   1:  PR[GP1:91,2] = PR[GP1:90,2] + -0.839;
   1:L PR[91] 10mm/sec CNT100;
   1:  PR[GP1:91,1] = PR[GP1:90,1] + 35.563;
   1:  PR[GP1:91,2] = PR[GP1:90,2] + -0.395;
   1:L PR[91] 10mm/sec CNT100;
   1:  PR[GP1:91,1] = PR[GP1:90,1] + 35.190;
   1:  PR[GP1:91,2] = PR[GP1:90,2] + 2.914;
   1:L PR[91] 10mm/sec CNT100;
   1:  PR[GP1:91,1] = PR[GP1:90,1] + 34.179;
   1:  PR[GP1:91,2] = PR[GP1:90,2] + 6.099;
   1:L PR[91] 10mm/sec CNT100;
   1:  PR[GP1:91,1] = PR[GP1:90,1] + 32.535;
   1:  PR[GP1:91,2] = PR[GP1:90,2] + 9.023;
   1:L PR[91] 10mm/sec CNT100;
   1:  PR[GP1:91,1] = PR[GP1:90,1] + 30.321;
   1:  PR[GP1:91,2] = PR[GP1:90,2] + 11.577;
   1:L PR[91] 10mm/sec CNT100;
   1:  PR[GP1:91,1] = PR[GP1:90,1] + 27.624;
   1:  PR[GP1:91,2] = PR[GP1:90,2] + 13.659;
   1:L PR[91] 10mm/sec CNT100;
   1:  PR[GP1:91,1] = PR[GP1:90,1] + 25.039;
   1:  PR[GP1:91,2] = PR[GP1:90,2] + 14.946;
   1:L PR[91] 10mm/sec CNT100;
   1:  PR[GP1:91,1] = PR[GP1:90,1] + 24.543;
   1:  PR[GP1:91,2] = PR[GP1:90,2] + 15.184;
   1:L PR[91] 10mm/sec CNT100;
   1:  PR[GP1:91,1] = PR[GP1:90,1] + 21.112;
   1:  PR[GP1:91,2] = PR[GP1:90,2] + 16.090;
   1:L PR[91] 10mm/sec CNT100;
   1:  PR[GP1:91,1] = PR[GP1:90,1] + 17.539;
   1:  PR[GP1:91,2] = PR[GP1:90,2] + 16.343;
   1:L PR[91] 10mm/sec CNT100;
   1:  PR[GP1:91,1] = PR[GP1:90,1] + 16.151;
   1:  PR[GP1:91,2] = PR[GP1:90,2] + 16.185;
   1:L PR[91] 10mm/sec CNT100;
   1:  PR[GP1:91,1] = PR[GP1:90,1] + 13.927;
   1:  PR[GP1:91,2] = PR[GP1:90,2] + 15.922;
   1:L PR[91] 10mm/sec CNT100;
   1:  PR[GP1:91,1] = PR[GP1:90,1] + 10.426;
   1:  PR[GP1:91,2] = PR[GP1:90,2] + 14.850;
   1:L PR[91] 10mm/sec CNT100;
   1:  PR[GP1:91,1] = PR[GP1:90,1] + 7.184;
   1:  PR[GP1:91,2] = PR[GP1:90,2] + 13.161;
   1:L PR[91] 10mm/sec CNT100;
   1:  PR[GP1:91,1] = PR[GP1:90,1] + 4.339;
   1:  PR[GP1:91,2] = PR[GP1:90,2] + 10.940;
   1:L PR[91] 10mm/sec CNT100;
   1:  PR[GP1:91,1] = PR[GP1:90,1] + 2.001;
   1:  PR[GP1:91,2] = PR[GP1:90,2] + 8.245;
   1:L PR[91] 10mm/sec CNT100;
   1:  PR[GP1:91,1] = PR[GP1:90,1] + 1.503;
   1:  PR[GP1:91,2] = PR[GP1:90,2] + 7.522;
   1:L PR[91] 10mm/sec CNT100;
   1:  PR[GP1:91,1] = PR[GP1:90,1] + 1.266;
   1:  PR[GP1:91,2] = PR[GP1:90,2] + 7.119;
   1:L PR[91] 10mm/sec CNT100;
   1:  PR[GP1:91,1] = PR[GP1:90,1] + 0.739;
   1:  PR[GP1:91,2] = PR[GP1:90,2] + 6.549;
   1:L PR[91] 10mm/sec CNT100;
   1:  PR[GP1:91,1] = PR[GP1:90,1] + 0.420;
   1:  PR[GP1:91,2] = PR[GP1:90,2] + 6.165;
   1:L PR[91] 10mm/sec CNT100;
   1:  PR[GP1:91,1] = PR[GP1:90,1] + -0.128;
   1:  PR[GP1:91,2] = PR[GP1:90,2] + 5.978;
   1:L PR[91] 10mm/sec CNT100;
   1:  PR[GP1:91,1] = PR[GP1:90,1] + -0.975;
   1:  PR[GP1:91,2] = PR[GP1:90,2] + 5.799;
   1:L PR[91] 10mm/sec CNT100;
   1:  PR[GP1:91,1] = PR[GP1:90,1] + -2.276;
   1:  PR[GP1:91,2] = PR[GP1:90,2] + 6.339;
   1:L PR[91] 10mm/sec CNT100;
   1:  PR[GP1:91,1] = PR[GP1:90,1] + -3.093;
   1:  PR[GP1:91,2] = PR[GP1:90,2] + 7.226;
   1:L PR[91] 10mm/sec CNT100;
   1:  PR[GP1:91,1] = PR[GP1:90,1] + -3.176;
   1:  PR[GP1:91,2] = PR[GP1:90,2] + 7.385;
   1:L PR[91] 10mm/sec CNT100;
   1:  PR[GP1:91,1] = PR[GP1:90,1] + -4.802;
   1:  PR[GP1:91,2] = PR[GP1:90,2] + 9.594;
   1:L PR[91] 10mm/sec CNT100;
   1:  PR[GP1:91,1] = PR[GP1:90,1] + -5.353;
   1:  PR[GP1:91,2] = PR[GP1:90,2] + 10.305;
   1:L PR[91] 10mm/sec CNT100;
   1:  PR[GP1:91,1] = PR[GP1:90,1] + -6.810;
   1:  PR[GP1:91,2] = PR[GP1:90,2] + 11.631;
   1:L PR[91] 10mm/sec CNT100;
   1:  PR[GP1:91,1] = PR[GP1:90,1] + -8.065;
   1:  PR[GP1:91,2] = PR[GP1:90,2] + 12.724;
   1:L PR[91] 10mm/sec CNT100;
   1:  PR[GP1:91,1] = PR[GP1:90,1] + -9.145;
   1:  PR[GP1:91,2] = PR[GP1:90,2] + 13.374;
   1:L PR[91] 10mm/sec CNT100;
   1:  PR[GP1:91,1] = PR[GP1:90,1] + -11.190;
   1:  PR[GP1:91,2] = PR[GP1:90,2] + 14.553;
   1:L PR[91] 10mm/sec CNT100;
   1:  PR[GP1:91,1] = PR[GP1:90,1] + -14.602;
   1:  PR[GP1:91,2] = PR[GP1:90,2] + 15.736;
   1:L PR[91] 10mm/sec CNT100;
   1:  PR[GP1:91,1] = PR[GP1:90,1] + -17.903;
   1:  PR[GP1:91,2] = PR[GP1:90,2] + 16.202;
   1:L PR[91] 10mm/sec CNT100;
   1:  PR[GP1:91,1] = PR[GP1:90,1] + -18.257;
   1:  PR[GP1:91,2] = PR[GP1:90,2] + 16.208;
   1:L PR[91] 10mm/sec CNT100;
   1:  PR[GP1:91,1] = PR[GP1:90,1] + -21.180;
   1:  PR[GP1:91,2] = PR[GP1:90,2] + 16.036;
   1:L PR[91] 10mm/sec CNT100;
   1:  PR[GP1:91,1] = PR[GP1:90,1] + -21.987;
   1:  PR[GP1:91,2] = PR[GP1:90,2] + 15.880;
   1:L PR[91] 10mm/sec CNT100;
   1:  PR[GP1:91,1] = PR[GP1:90,1] + -24.427;
   1:  PR[GP1:91,2] = PR[GP1:90,2] + 15.235;
   1:L PR[91] 10mm/sec CNT100;
   1:  PR[GP1:91,1] = PR[GP1:90,1] + -25.526;
   1:  PR[GP1:91,2] = PR[GP1:90,2] + 14.770;
   1:L PR[91] 10mm/sec CNT100;
   1:  PR[GP1:91,1] = PR[GP1:90,1] + -27.498;
   1:  PR[GP1:91,2] = PR[GP1:90,2] + 13.796;
   1:L PR[91] 10mm/sec CNT100;
   1:  PR[GP1:91,1] = PR[GP1:90,1] + -28.704;
   1:  PR[GP1:91,2] = PR[GP1:90,2] + 12.949;
   1:L PR[91] 10mm/sec CNT100;
   1:  PR[GP1:91,1] = PR[GP1:90,1] + -30.246;
   1:  PR[GP1:91,2] = PR[GP1:90,2] + 11.752;
   1:L PR[91] 10mm/sec CNT100;
   1:  PR[GP1:91,1] = PR[GP1:90,1] + -31.379;
   1:  PR[GP1:91,2] = PR[GP1:90,2] + 10.524;
   1:L PR[91] 10mm/sec CNT100;
   1:  PR[GP1:91,1] = PR[GP1:90,1] + -32.532;
   1:  PR[GP1:91,2] = PR[GP1:90,2] + 9.173;
   1:L PR[91] 10mm/sec CNT100;
   1:  PR[GP1:91,1] = PR[GP1:90,1] + -33.440;
   1:  PR[GP1:91,2] = PR[GP1:90,2] + 7.630;
   1:L PR[91] 10mm/sec CNT100;
   1:  PR[GP1:91,1] = PR[GP1:90,1] + -34.248;
   1:  PR[GP1:91,2] = PR[GP1:90,2] + 6.164;
   1:L PR[91] 10mm/sec CNT100;
   1:  PR[GP1:91,1] = PR[GP1:90,1] + -34.824;
   1:  PR[GP1:91,2] = PR[GP1:90,2] + 4.418;
   1:L PR[91] 10mm/sec CNT100;
   1:  PR[GP1:91,1] = PR[GP1:90,1] + -35.313;
   1:  PR[GP1:91,2] = PR[GP1:90,2] + 2.861;
   1:L PR[91] 10mm/sec CNT100;
   1:  PR[GP1:91,1] = PR[GP1:90,1] + -35.500;
   1:  PR[GP1:91,2] = PR[GP1:90,2] + 1.034;
   1:L PR[91] 10mm/sec CNT100;
   1:  PR[GP1:91,1] = PR[GP1:90,1] + -35.737;
   1:  PR[GP1:91,2] = PR[GP1:90,2] + -0.426;
   1:L PR[91] 10mm/sec CNT100;
   1:  PR[GP1:91,1] = PR[GP1:90,1] + -35.748;
   1:  PR[GP1:91,2] = PR[GP1:90,2] + -0.547;
   1:L PR[91] 10mm/sec CNT100;
   1:  PR[GP1:91,1] = PR[GP1:90,1] + -35.460;
   1:  PR[GP1:91,2] = PR[GP1:90,2] + -2.299;
   1:L PR[91] 10mm/sec CNT100;
   1:  PR[GP1:91,1] = PR[GP1:90,1] + -35.263;
   1:  PR[GP1:91,2] = PR[GP1:90,2] + -4.065;
   1:L PR[91] 10mm/sec CNT100;
   1:  PR[GP1:91,1] = PR[GP1:90,1] + -34.667;
   1:  PR[GP1:91,2] = PR[GP1:90,2] + -5.939;
   1:L PR[91] 10mm/sec CNT100;
   1:  PR[GP1:91,1] = PR[GP1:90,1] + -34.192;
   1:  PR[GP1:91,2] = PR[GP1:90,2] + -7.356;
   1:L PR[91] 10mm/sec CNT100;
   1:  PR[GP1:91,1] = PR[GP1:90,1] + -33.095;
   1:  PR[GP1:91,2] = PR[GP1:90,2] + -9.301;
   1:L PR[91] 10mm/sec CNT100;
   1:  PR[GP1:91,1] = PR[GP1:90,1] + -32.472;
   1:  PR[GP1:91,2] = PR[GP1:90,2] + -10.348;
   1:L PR[91] 10mm/sec CNT100;
   1:  PR[GP1:91,1] = PR[GP1:90,1] + -30.781;
   1:  PR[GP1:91,2] = PR[GP1:90,2] + -12.296;
   1:L PR[91] 10mm/sec CNT100;
   1:  PR[GP1:91,1] = PR[GP1:90,1] + -30.208;
   1:  PR[GP1:91,2] = PR[GP1:90,2] + -12.915;
   1:L PR[91] 10mm/sec CNT100;
   1:  PR[GP1:91,1] = PR[GP1:90,1] + -27.823;
   1:  PR[GP1:91,2] = PR[GP1:90,2] + -14.750;
   1:L PR[91] 10mm/sec CNT100;
   1:  PR[GP1:91,1] = PR[GP1:90,1] + -27.525;
   1:  PR[GP1:91,2] = PR[GP1:90,2] + -14.960;
   1:L PR[91] 10mm/sec CNT100;
   1:  PR[GP1:91,1] = PR[GP1:90,1] + -24.458;
   1:  PR[GP1:91,2] = PR[GP1:90,2] + -16.461;
   1:L PR[91] 10mm/sec CNT100;
   1:  PR[GP1:91,1] = PR[GP1:90,1] + -24.049;
   1:  PR[GP1:91,2] = PR[GP1:90,2] + -16.598;
   1:  PR[GP1:91,3] = PR[GP1:90,3] + 16.500;
   1:L PR[91] 10mm/sec CNT100;
   1:  PR[GP1:91,1] = PR[GP1:90,1] + -21.809;
   1:  PR[GP1:91,2] = PR[GP1:90,2] + -17.202;
   1:L PR[91] 10mm/sec CNT100;
   1:  PR[GP1:91,1] = PR[GP1:90,1] + -20.477;
   1:  PR[GP1:91,2] = PR[GP1:90,2] + -17.522;
   1:L PR[91] 10mm/sec CNT100;
   1:  PR[GP1:91,1] = PR[GP1:90,1] + -18.846;
   1:  PR[GP1:91,2] = PR[GP1:90,2] + -17.637;
   1:L PR[91] 10mm/sec CNT100;
   1:  PR[GP1:91,1] = PR[GP1:90,1] + -16.756;
   1:  PR[GP1:91,2] = PR[GP1:90,2] + -17.718;
   1:L PR[91] 10mm/sec CNT100;
   1:  PR[GP1:91,1] = PR[GP1:90,1] + -15.910;
   1:  PR[GP1:91,2] = PR[GP1:90,2] + -17.613;
   1:L PR[91] 10mm/sec CNT100;
   1:  PR[GP1:91,1] = PR[GP1:90,1] + -13.050;
   1:  PR[GP1:91,2] = PR[GP1:90,2] + -17.151;
   1:L PR[91] 10mm/sec CNT100;
   1:  PR[GP1:91,1] = PR[GP1:90,1] + -10.065;
   1:  PR[GP1:91,2] = PR[GP1:90,2] + -16.120;
   1:L PR[91] 10mm/sec CNT100;
   1:  PR[GP1:91,1] = PR[GP1:90,1] + -9.281;
   1:  PR[GP1:91,2] = PR[GP1:90,2] + -15.790;
   1:L PR[91] 10mm/sec CNT100;
   1:  PR[GP1:91,1] = PR[GP1:90,1] + -7.395;
   1:  PR[GP1:91,2] = PR[GP1:90,2] + -14.673;
   1:L PR[91] 10mm/sec CNT100;
   1:  PR[GP1:91,1] = PR[GP1:90,1] + -5.918;
   1:  PR[GP1:91,2] = PR[GP1:90,2] + -13.640;
   1:L PR[91] 10mm/sec CNT100;
   1:  PR[GP1:91,1] = PR[GP1:90,1] + -5.000;
   1:  PR[GP1:91,2] = PR[GP1:90,2] + -12.787;
   1:L PR[91] 10mm/sec CNT100;
   1:  PR[GP1:91,1] = PR[GP1:90,1] + -3.184;
   1:  PR[GP1:91,2] = PR[GP1:90,2] + -10.770;
   1:L PR[91] 10mm/sec CNT100;
   1:  PR[GP1:91,1] = PR[GP1:90,1] + -2.909;
   1:  PR[GP1:91,2] = PR[GP1:90,2] + -10.366;
   1:L PR[91] 10mm/sec CNT100;
   1:  PR[GP1:91,1] = PR[GP1:90,1] + -2.225;
   1:  PR[GP1:91,2] = PR[GP1:90,2] + -9.700;
   1:L PR[91] 10mm/sec CNT100;
   1:  PR[GP1:91,1] = PR[GP1:90,1] + -1.965;
   1:  PR[GP1:91,2] = PR[GP1:90,2] + -9.545;
   1:L PR[91] 10mm/sec CNT100;
   1:  PR[GP1:91,1] = PR[GP1:90,1] + -1.033;
   1:  PR[GP1:91,2] = PR[GP1:90,2] + -9.287;
   1:L PR[91] 10mm/sec CNT100;
   1:  PR[GP1:91,1] = PR[GP1:90,1] + -0.752;
   1:  PR[GP1:91,2] = PR[GP1:90,2] + -9.306;
   1:L PR[91] 10mm/sec CNT100;
   1:  PR[GP1:91,1] = PR[GP1:90,1] + 0.181;
   1:  PR[GP1:91,2] = PR[GP1:90,2] + -9.570;
   1:L PR[91] 10mm/sec CNT100;
   1:  PR[GP1:91,1] = PR[GP1:90,1] + 0.446;
   1:  PR[GP1:91,2] = PR[GP1:90,2] + -9.766;
   1:L PR[91] 10mm/sec CNT100;
   1:  PR[GP1:91,1] = PR[GP1:90,1] + 1.063;
   1:  PR[GP1:91,2] = PR[GP1:90,2] + -10.427;
   1:L PR[91] 10mm/sec CNT100;
   1:  PR[GP1:91,1] = PR[GP1:90,1] + 1.209;
   1:  PR[GP1:91,2] = PR[GP1:90,2] + -10.623;
   1:L PR[91] 10mm/sec CNT100;
   1:  PR[GP1:91,1] = PR[GP1:90,1] + 2.802;
   1:  PR[GP1:91,2] = PR[GP1:90,2] + -12.531;
   1:L PR[91] 10mm/sec CNT100;
   1:  PR[GP1:91,1] = PR[GP1:90,1] + 3.060;
   1:  PR[GP1:91,2] = PR[GP1:90,2] + -12.778;
   1:L PR[91] 10mm/sec CNT100;
   1:  PR[GP1:91,1] = PR[GP1:90,1] + 4.730;
   1:  PR[GP1:91,2] = PR[GP1:90,2] + -14.227;
   1:L PR[91] 10mm/sec CNT100;
   1:  PR[GP1:91,1] = PR[GP1:90,1] + 5.384;
   1:  PR[GP1:91,2] = PR[GP1:90,2] + -14.675;
   1:L PR[91] 10mm/sec CNT100;
   1:  PR[GP1:91,1] = PR[GP1:90,1] + 6.911;
   1:  PR[GP1:91,2] = PR[GP1:90,2] + -15.628;
   1:L PR[91] 10mm/sec CNT100;
   1:  PR[GP1:91,1] = PR[GP1:90,1] + 8.184;
   1:  PR[GP1:91,2] = PR[GP1:90,2] + -16.230;
   1:L PR[91] 10mm/sec CNT100;
   1:  PR[GP1:91,1] = PR[GP1:90,1] + 9.302;
   1:  PR[GP1:91,2] = PR[GP1:90,2] + -16.710;
   1:L PR[91] 10mm/sec CNT100;
   1:  PR[GP1:91,1] = PR[GP1:90,1] + 11.435;
   1:  PR[GP1:91,2] = PR[GP1:90,2] + -17.342;
   1:L PR[91] 10mm/sec CNT100;
   1:  PR[GP1:91,1] = PR[GP1:90,1] + 11.858;
   1:  PR[GP1:91,2] = PR[GP1:90,2] + -17.453;
   1:L PR[91] 10mm/sec CNT100;
   1:  PR[GP1:91,1] = PR[GP1:90,1] + 13.231;
   1:  PR[GP1:91,2] = PR[GP1:90,2] + -17.645;
   1:L PR[91] 10mm/sec CNT100;
   1:  PR[GP1:91,1] = PR[GP1:90,1] + 14.565;
   1:  PR[GP1:91,2] = PR[GP1:90,2] + -17.853;
   1:L PR[91] 10mm/sec CNT100;
   1:  PR[GP1:91,1] = PR[GP1:90,1] + 17.338;
   1:  PR[GP1:91,2] = PR[GP1:90,2] + -17.894;
   1:L PR[91] 10mm/sec CNT100;
   1:  PR[GP1:91,1] = PR[GP1:90,1] + 20.128;
   1:  PR[GP1:91,2] = PR[GP1:90,2] + -17.557;
   1:L PR[91] 10mm/sec CNT100;
   1:  PR[GP1:91,1] = PR[GP1:90,1] + 22.900;
   1:  PR[GP1:91,2] = PR[GP1:90,2] + -16.831;
   1:L PR[91] 10mm/sec CNT100;
   1:  PR[GP1:91,1] = PR[GP1:90,1] + 25.555;
   1:  PR[GP1:91,2] = PR[GP1:90,2] + -15.714;
   1:L PR[91] 10mm/sec CNT100;
   1:  PR[GP1:91,1] = PR[GP1:90,1] + 27.990;
   1:  PR[GP1:91,2] = PR[GP1:90,2] + -14.238;
   1:L PR[91] 10mm/sec CNT100;
   1:  PR[GP1:91,1] = PR[GP1:90,1] + 30.137;
   1:  PR[GP1:91,2] = PR[GP1:90,2] + -12.447;
   1:L PR[91] 10mm/sec CNT100;
   1:  PR[GP1:91,1] = PR[GP1:90,1] + 31.915;
   1:  PR[GP1:91,2] = PR[GP1:90,2] + -10.393;
   1:L PR[91] 10mm/sec CNT100;
   1:  PR[GP1:91,1] = PR[GP1:90,1] + 33.342;
   1:  PR[GP1:91,2] = PR[GP1:90,2] + -8.106;
   1:L PR[91] 10mm/sec CNT100;
   1:  PR[GP1:91,1] = PR[GP1:90,1] + 34.386;
   1:  PR[GP1:91,2] = PR[GP1:90,2] + -5.644;
   1:L PR[91] 10mm/sec CNT100;
   1:  PR[GP1:91,1] = PR[GP1:90,1] + 35.021;
   1:  PR[GP1:91,2] = PR[GP1:90,2] + -3.065;
   1:L PR[91] 10mm/sec CNT100;
   1:  PR[GP1:91,1] = PR[GP1:90,1] + 35.141;
   1:  PR[GP1:91,2] = PR[GP1:90,2] + -1.599;
   1:L PR[91] 10mm/sec CNT100;
   1:  PR[GP1:91,1] = PR[GP1:90,1] + 35.273;
   1:  PR[GP1:91,2] = PR[GP1:90,2] + -0.425;
   1:L PR[91] 10mm/sec CNT100;
   1:  PR[GP1:91,1] = PR[GP1:90,1] + 34.888;
   1:  PR[GP1:91,2] = PR[GP1:90,2] + 2.885;
   1:L PR[91] 10mm/sec CNT100;
   1:  PR[GP1:91,1] = PR[GP1:90,1] + 33.871;
   1:  PR[GP1:91,2] = PR[GP1:90,2] + 6.072;
   1:L PR[91] 10mm/sec CNT100;
   1:  PR[GP1:91,1] = PR[GP1:90,1] + 32.223;
   1:  PR[GP1:91,2] = PR[GP1:90,2] + 8.997;
   1:L PR[91] 10mm/sec CNT100;
   1:  PR[GP1:91,1] = PR[GP1:90,1] + 30.005;
   1:  PR[GP1:91,2] = PR[GP1:90,2] + 11.551;
   1:L PR[91] 10mm/sec CNT100;
   1:  PR[GP1:91,1] = PR[GP1:90,1] + 28.164;
   1:  PR[GP1:91,2] = PR[GP1:90,2] + 12.971;
   1:L PR[91] 10mm/sec CNT100;
   1:  PR[GP1:91,1] = PR[GP1:90,1] + 27.290;
   1:  PR[GP1:91,2] = PR[GP1:90,2] + 13.625;
   1:L PR[91] 10mm/sec CNT100;
   1:  PR[GP1:91,1] = PR[GP1:90,1] + 24.125;
   1:  PR[GP1:91,2] = PR[GP1:90,2] + 15.144;
   1:L PR[91] 10mm/sec CNT100;
   1:  PR[GP1:91,1] = PR[GP1:90,1] + 20.701;
   1:  PR[GP1:91,2] = PR[GP1:90,2] + 16.048;
   1:L PR[91] 10mm/sec CNT100;
   1:  PR[GP1:91,1] = PR[GP1:90,1] + 17.093;
   1:  PR[GP1:91,2] = PR[GP1:90,2] + 16.290;
   1:L PR[91] 10mm/sec CNT100;
   1:  PR[GP1:91,1] = PR[GP1:90,1] + 13.444;
   1:  PR[GP1:91,2] = PR[GP1:90,2] + 15.859;
   1:L PR[91] 10mm/sec CNT100;
   1:  PR[GP1:91,1] = PR[GP1:90,1] + 9.932;
   1:  PR[GP1:91,2] = PR[GP1:90,2] + 14.773;
   1:L PR[91] 10mm/sec CNT100;
   1:  PR[GP1:91,1] = PR[GP1:90,1] + 6.681;
   1:  PR[GP1:91,2] = PR[GP1:90,2] + 13.083;
   1:L PR[91] 10mm/sec CNT100;
   1:  PR[GP1:91,1] = PR[GP1:90,1] + 3.849;
   1:  PR[GP1:91,2] = PR[GP1:90,2] + 10.848;
   1:L PR[91] 10mm/sec CNT100;
   1:  PR[GP1:91,1] = PR[GP1:90,1] + 1.504;
   1:  PR[GP1:91,2] = PR[GP1:90,2] + 8.159;
   1:L PR[91] 10mm/sec CNT100;
   1:  PR[GP1:91,1] = PR[GP1:90,1] + 1.159;
   1:  PR[GP1:91,2] = PR[GP1:90,2] + 7.659;
   1:L PR[91] 10mm/sec CNT100;
   1:  PR[GP1:91,1] = PR[GP1:90,1] + 0.530;
   1:  PR[GP1:91,2] = PR[GP1:90,2] + 7.106;
   1:L PR[91] 10mm/sec CNT100;
   1:  PR[GP1:91,1] = PR[GP1:90,1] + 0.267;
   1:  PR[GP1:91,2] = PR[GP1:90,2] + 6.814;
   1:L PR[91] 10mm/sec CNT100;
   1:  PR[GP1:91,1] = PR[GP1:90,1] + -1.097;
   1:  PR[GP1:91,2] = PR[GP1:90,2] + 6.515;
   1:L PR[91] 10mm/sec CNT100;
   1:  PR[GP1:91,1] = PR[GP1:90,1] + -1.473;
   1:  PR[GP1:91,2] = PR[GP1:90,2] + 6.676;
   1:L PR[91] 10mm/sec CNT100;
   1:  PR[GP1:91,1] = PR[GP1:90,1] + -2.323;
   1:  PR[GP1:91,2] = PR[GP1:90,2] + 6.945;
   1:L PR[91] 10mm/sec CNT100;
   1:  PR[GP1:91,1] = PR[GP1:90,1] + -3.014;
   1:  PR[GP1:91,2] = PR[GP1:90,2] + 7.674;
   1:L PR[91] 10mm/sec CNT100;
   1:  PR[GP1:91,1] = PR[GP1:90,1] + -4.937;
   1:  PR[GP1:91,2] = PR[GP1:90,2] + 10.131;
   1:L PR[91] 10mm/sec CNT100;
   1:  PR[GP1:91,1] = PR[GP1:90,1] + -7.022;
   1:  PR[GP1:91,2] = PR[GP1:90,2] + 12.028;
   1:L PR[91] 10mm/sec CNT100;
   1:  PR[GP1:91,1] = PR[GP1:90,1] + -7.655;
   1:  PR[GP1:91,2] = PR[GP1:90,2] + 12.579;
   1:L PR[91] 10mm/sec CNT100;
   1:  PR[GP1:91,1] = PR[GP1:90,1] + -9.399;
   1:  PR[GP1:91,2] = PR[GP1:90,2] + 13.630;
   1:L PR[91] 10mm/sec CNT100;
   1:  PR[GP1:91,1] = PR[GP1:90,1] + -10.792;
   1:  PR[GP1:91,2] = PR[GP1:90,2] + 14.432;
   1:L PR[91] 10mm/sec CNT100;
   1:  PR[GP1:91,1] = PR[GP1:90,1] + -12.052;
   1:  PR[GP1:91,2] = PR[GP1:90,2] + 14.889;
   1:L PR[91] 10mm/sec CNT100;
   1:  PR[GP1:91,1] = PR[GP1:90,1] + -14.210;
   1:  PR[GP1:91,2] = PR[GP1:90,2] + 15.629;
   1:L PR[91] 10mm/sec CNT100;
   1:  PR[GP1:91,1] = PR[GP1:90,1] + -17.771;
   1:  PR[GP1:91,2] = PR[GP1:90,2] + 16.139;
   1:L PR[91] 10mm/sec CNT100;
   1:  PR[GP1:91,1] = PR[GP1:90,1] + -21.225;
   1:  PR[GP1:91,2] = PR[GP1:90,2] + 15.950;
   1:L PR[91] 10mm/sec CNT100;
   1:  PR[GP1:91,1] = PR[GP1:90,1] + -21.354;
   1:  PR[GP1:91,2] = PR[GP1:90,2] + 15.925;
   1:L PR[91] 10mm/sec CNT100;
   1:  PR[GP1:91,1] = PR[GP1:90,1] + -24.418;
   1:  PR[GP1:91,2] = PR[GP1:90,2] + 15.116;
   1:L PR[91] 10mm/sec CNT100;
   1:  PR[GP1:91,1] = PR[GP1:90,1] + -24.918;
   1:  PR[GP1:91,2] = PR[GP1:90,2] + 14.903;
   1:L PR[91] 10mm/sec CNT100;
   1:  PR[GP1:91,1] = PR[GP1:90,1] + -27.439;
   1:  PR[GP1:91,2] = PR[GP1:90,2] + 13.659;
   1:L PR[91] 10mm/sec CNT100;
   1:  PR[GP1:91,1] = PR[GP1:90,1] + -28.140;
   1:  PR[GP1:91,2] = PR[GP1:90,2] + 13.167;
   1:L PR[91] 10mm/sec CNT100;
   1:  PR[GP1:91,1] = PR[GP1:90,1] + -30.142;
   1:  PR[GP1:91,2] = PR[GP1:90,2] + 11.612;
   1:L PR[91] 10mm/sec CNT100;
   1:  PR[GP1:91,1] = PR[GP1:90,1] + -30.873;
   1:  PR[GP1:91,2] = PR[GP1:90,2] + 10.820;
   1:L PR[91] 10mm/sec CNT100;
   1:  PR[GP1:91,1] = PR[GP1:90,1] + -32.392;
   1:  PR[GP1:91,2] = PR[GP1:90,2] + 9.041;
   1:L PR[91] 10mm/sec CNT100;
   1:  PR[GP1:91,1] = PR[GP1:90,1] + -33.008;
   1:  PR[GP1:91,2] = PR[GP1:90,2] + 7.994;
   1:L PR[91] 10mm/sec CNT100;
   1:  PR[GP1:91,1] = PR[GP1:90,1] + -34.079;
   1:  PR[GP1:91,2] = PR[GP1:90,2] + 6.050;
   1:L PR[91] 10mm/sec CNT100;
   1:  PR[GP1:91,1] = PR[GP1:90,1] + -34.479;
   1:  PR[GP1:91,2] = PR[GP1:90,2] + 4.838;
   1:L PR[91] 10mm/sec CNT100;
   1:  PR[GP1:91,1] = PR[GP1:90,1] + -35.129;
   1:  PR[GP1:91,2] = PR[GP1:90,2] + 2.771;
   1:L PR[91] 10mm/sec CNT100;
   1:  PR[GP1:91,1] = PR[GP1:90,1] + -35.259;
   1:  PR[GP1:91,2] = PR[GP1:90,2] + 1.496;
   1:L PR[91] 10mm/sec CNT100;
   1:  PR[GP1:91,1] = PR[GP1:90,1] + -35.426;
   1:  PR[GP1:91,2] = PR[GP1:90,2] + 0.467;
   1:L PR[91] 10mm/sec CNT100;
   1:  PR[GP1:91,1] = PR[GP1:90,1] + -35.526;
   1:  PR[GP1:91,2] = PR[GP1:90,2] + -0.621;
   1:L PR[91] 10mm/sec CNT100;
   1:  PR[GP1:91,1] = PR[GP1:90,1] + -35.330;
   1:  PR[GP1:91,2] = PR[GP1:90,2] + -1.808;
   1:L PR[91] 10mm/sec CNT100;
   1:  PR[GP1:91,1] = PR[GP1:90,1] + -35.074;
   1:  PR[GP1:91,2] = PR[GP1:90,2] + -4.102;
   1:L PR[91] 10mm/sec CNT100;
   1:  PR[GP1:91,1] = PR[GP1:90,1] + -34.300;
   1:  PR[GP1:91,2] = PR[GP1:90,2] + -6.541;
   1:L PR[91] 10mm/sec CNT100;
   1:  PR[GP1:91,1] = PR[GP1:90,1] + -34.023;
   1:  PR[GP1:91,2] = PR[GP1:90,2] + -7.366;
   1:L PR[91] 10mm/sec CNT100;
   1:  PR[GP1:91,1] = PR[GP1:90,1] + -32.618;
   1:  PR[GP1:91,2] = PR[GP1:90,2] + -9.858;
   1:L PR[91] 10mm/sec CNT100;
   1:  PR[GP1:91,1] = PR[GP1:90,1] + -32.333;
   1:  PR[GP1:91,2] = PR[GP1:90,2] + -10.338;
   1:L PR[91] 10mm/sec CNT100;
   1:  PR[GP1:91,1] = PR[GP1:90,1] + -30.204;
   1:  PR[GP1:91,2] = PR[GP1:90,2] + -12.789;
   1:L PR[91] 10mm/sec CNT100;
   1:  PR[GP1:91,1] = PR[GP1:90,1] + -30.110;
   1:  PR[GP1:91,2] = PR[GP1:90,2] + -12.891;
   1:L PR[91] 10mm/sec CNT100;
   1:  PR[GP1:91,1] = PR[GP1:90,1] + -27.320;
   1:  PR[GP1:91,2] = PR[GP1:90,2] + -15.014;
   1:L PR[91] 10mm/sec CNT100;
   1:  PR[GP1:91,1] = PR[GP1:90,1] + -24.722;
   1:  PR[GP1:91,2] = PR[GP1:90,2] + -16.288;
   1:L PR[91] 10mm/sec CNT100;
   1:  PR[GP1:91,1] = PR[GP1:90,1] + -23.632;
   1:  PR[GP1:91,2] = PR[GP1:90,2] + -16.737;
   1:  PR[GP1:91,3] = PR[GP1:90,3] + 17.600;
   1:L PR[91] 10mm/sec CNT100;
   1:  PR[GP1:91,1] = PR[GP1:90,1] + -22.073;
   1:  PR[GP1:91,2] = PR[GP1:90,2] + -17.157;
   1:L PR[91] 10mm/sec CNT100;
   1:  PR[GP1:91,1] = PR[GP1:90,1] + -20.031;
   1:  PR[GP1:91,2] = PR[GP1:90,2] + -17.648;
   1:L PR[91] 10mm/sec CNT100;
   1:  PR[GP1:91,1] = PR[GP1:90,1] + -19.162;
   1:  PR[GP1:91,2] = PR[GP1:90,2] + -17.710;
   1:L PR[91] 10mm/sec CNT100;
   1:  PR[GP1:91,1] = PR[GP1:90,1] + -16.282;
   1:  PR[GP1:91,2] = PR[GP1:90,2] + -17.821;
   1:L PR[91] 10mm/sec CNT100;
   1:  PR[GP1:91,1] = PR[GP1:90,1] + -13.121;
   1:  PR[GP1:91,2] = PR[GP1:90,2] + -17.389;
   1:L PR[91] 10mm/sec CNT100;
   1:  PR[GP1:91,1] = PR[GP1:90,1] + -12.278;
   1:  PR[GP1:91,2] = PR[GP1:90,2] + -17.222;
   1:L PR[91] 10mm/sec CNT100;
   1:  PR[GP1:91,1] = PR[GP1:90,1] + -10.225;
   1:  PR[GP1:91,2] = PR[GP1:90,2] + -16.518;
   1:L PR[91] 10mm/sec CNT100;
   1:  PR[GP1:91,1] = PR[GP1:90,1] + -8.447;
   1:  PR[GP1:91,2] = PR[GP1:90,2] + -15.769;
   1:L PR[91] 10mm/sec CNT100;
   1:  PR[GP1:91,1] = PR[GP1:90,1] + -7.521;
   1:  PR[GP1:91,2] = PR[GP1:90,2] + -15.220;
   1:L PR[91] 10mm/sec CNT100;
   1:  PR[GP1:91,1] = PR[GP1:90,1] + -5.098;
   1:  PR[GP1:91,2] = PR[GP1:90,2] + -13.526;
   1:L PR[91] 10mm/sec CNT100;
   1:  PR[GP1:91,1] = PR[GP1:90,1] + -4.779;
   1:  PR[GP1:91,2] = PR[GP1:90,2] + -13.184;
   1:L PR[91] 10mm/sec CNT100;
   1:  PR[GP1:91,1] = PR[GP1:90,1] + -2.747;
   1:  PR[GP1:91,2] = PR[GP1:90,2] + -11.110;
   1:L PR[91] 10mm/sec CNT100;
   1:  PR[GP1:91,1] = PR[GP1:90,1] + -2.284;
   1:  PR[GP1:91,2] = PR[GP1:90,2] + -10.666;
   1:L PR[91] 10mm/sec CNT100;
   1:  PR[GP1:91,1] = PR[GP1:90,1] + -1.776;
   1:  PR[GP1:91,2] = PR[GP1:90,2] + -10.363;
   1:L PR[91] 10mm/sec CNT100;
   1:  PR[GP1:91,1] = PR[GP1:90,1] + -1.082;
   1:  PR[GP1:91,2] = PR[GP1:90,2] + -10.171;
   1:L PR[91] 10mm/sec CNT100;
   1:  PR[GP1:91,1] = PR[GP1:90,1] + -0.525;
   1:  PR[GP1:91,2] = PR[GP1:90,2] + -10.209;
   1:L PR[91] 10mm/sec CNT100;
   1:  PR[GP1:91,1] = PR[GP1:90,1] + 0.158;
   1:  PR[GP1:91,2] = PR[GP1:90,2] + -10.402;
   1:L PR[91] 10mm/sec CNT100;
   1:  PR[GP1:91,1] = PR[GP1:90,1] + 0.712;
   1:  PR[GP1:91,2] = PR[GP1:90,2] + -10.812;
   1:L PR[91] 10mm/sec CNT100;
   1:  PR[GP1:91,1] = PR[GP1:90,1] + 0.851;
   1:  PR[GP1:91,2] = PR[GP1:90,2] + -11.005;
   1:L PR[91] 10mm/sec CNT100;
   1:  PR[GP1:91,1] = PR[GP1:90,1] + 1.058;
   1:  PR[GP1:91,2] = PR[GP1:90,2] + -11.227;
   1:L PR[91] 10mm/sec CNT100;
   1:  PR[GP1:91,1] = PR[GP1:90,1] + 2.039;
   1:  PR[GP1:91,2] = PR[GP1:90,2] + -12.391;
   1:L PR[91] 10mm/sec CNT100;
   1:  PR[GP1:91,1] = PR[GP1:90,1] + 2.398;
   1:  PR[GP1:91,2] = PR[GP1:90,2] + -12.782;
   1:L PR[91] 10mm/sec CNT100;
   1:  PR[GP1:91,1] = PR[GP1:90,1] + 4.390;
   1:  PR[GP1:91,2] = PR[GP1:90,2] + -14.508;
   1:L PR[91] 10mm/sec CNT100;
   1:  PR[GP1:91,1] = PR[GP1:90,1] + 6.605;
   1:  PR[GP1:91,2] = PR[GP1:90,2] + -15.893;
   1:L PR[91] 10mm/sec CNT100;
   1:  PR[GP1:91,1] = PR[GP1:90,1] + 7.051;
   1:  PR[GP1:91,2] = PR[GP1:90,2] + -16.104;
   1:L PR[91] 10mm/sec CNT100;
   1:  PR[GP1:91,1] = PR[GP1:90,1] + 9.006;
   1:  PR[GP1:91,2] = PR[GP1:90,2] + -16.943;
   1:L PR[91] 10mm/sec CNT100;
   1:  PR[GP1:91,1] = PR[GP1:90,1] + 10.197;
   1:  PR[GP1:91,2] = PR[GP1:90,2] + -17.296;
   1:L PR[91] 10mm/sec CNT100;
   1:  PR[GP1:91,1] = PR[GP1:90,1] + 11.566;
   1:  PR[GP1:91,2] = PR[GP1:90,2] + -17.656;
   1:L PR[91] 10mm/sec CNT100;
   1:  PR[GP1:91,1] = PR[GP1:90,1] + 13.741;
   1:  PR[GP1:91,2] = PR[GP1:90,2] + -17.960;
   1:L PR[91] 10mm/sec CNT100;
   1:  PR[GP1:91,1] = PR[GP1:90,1] + 14.236;
   1:  PR[GP1:91,2] = PR[GP1:90,2] + -18.015;
   1:L PR[91] 10mm/sec CNT100;
   1:  PR[GP1:91,1] = PR[GP1:90,1] + 15.625;
   1:  PR[GP1:91,2] = PR[GP1:90,2] + -18.006;
   1:L PR[91] 10mm/sec CNT100;
   1:  PR[GP1:91,1] = PR[GP1:90,1] + 17.004;
   1:  PR[GP1:91,2] = PR[GP1:90,2] + -18.020;
   1:L PR[91] 10mm/sec CNT100;
   1:  PR[GP1:91,1] = PR[GP1:90,1] + 19.780;
   1:  PR[GP1:91,2] = PR[GP1:90,2] + -17.663;
   1:L PR[91] 10mm/sec CNT100;
   1:  PR[GP1:91,1] = PR[GP1:90,1] + 22.509;
   1:  PR[GP1:91,2] = PR[GP1:90,2] + -16.928;
   1:L PR[91] 10mm/sec CNT100;
   1:  PR[GP1:91,1] = PR[GP1:90,1] + 25.143;
   1:  PR[GP1:91,2] = PR[GP1:90,2] + -15.812;
   1:L PR[91] 10mm/sec CNT100;
   1:  PR[GP1:91,1] = PR[GP1:90,1] + 27.585;
   1:  PR[GP1:91,2] = PR[GP1:90,2] + -14.329;
   1:L PR[91] 10mm/sec CNT100;
   1:  PR[GP1:91,1] = PR[GP1:90,1] + 29.750;
   1:  PR[GP1:91,2] = PR[GP1:90,2] + -12.524;
   1:L PR[91] 10mm/sec CNT100;
   1:  PR[GP1:91,1] = PR[GP1:90,1] + 31.588;
   1:  PR[GP1:91,2] = PR[GP1:90,2] + -10.446;
   1:L PR[91] 10mm/sec CNT100;
   1:  PR[GP1:91,1] = PR[GP1:90,1] + 33.034;
   1:  PR[GP1:91,2] = PR[GP1:90,2] + -8.151;
   1:L PR[91] 10mm/sec CNT100;
   1:  PR[GP1:91,1] = PR[GP1:90,1] + 34.075;
   1:  PR[GP1:91,2] = PR[GP1:90,2] + -5.686;
   1:L PR[91] 10mm/sec CNT100;
   1:  PR[GP1:91,1] = PR[GP1:90,1] + 34.708;
   1:  PR[GP1:91,2] = PR[GP1:90,2] + -3.102;
   1:L PR[91] 10mm/sec CNT100;
   1:  PR[GP1:91,1] = PR[GP1:90,1] + 34.769;
   1:  PR[GP1:91,2] = PR[GP1:90,2] + -2.359;
   1:L PR[91] 10mm/sec CNT100;
   1:  PR[GP1:91,1] = PR[GP1:90,1] + 34.868;
   1:  PR[GP1:91,2] = PR[GP1:90,2] + -1.475;
   1:L PR[91] 10mm/sec CNT100;
   1:  PR[GP1:91,1] = PR[GP1:90,1] + 34.947;
   1:  PR[GP1:91,2] = PR[GP1:90,2] + -0.465;
   1:L PR[91] 10mm/sec CNT100;
   1:  PR[GP1:91,1] = PR[GP1:90,1] + 34.749;
   1:  PR[GP1:91,2] = PR[GP1:90,2] + 1.466;
   1:L PR[91] 10mm/sec CNT100;
   1:  PR[GP1:91,1] = PR[GP1:90,1] + 34.585;
   1:  PR[GP1:91,2] = PR[GP1:90,2] + 2.856;
   1:L PR[91] 10mm/sec CNT100;
   1:  PR[GP1:91,1] = PR[GP1:90,1] + 33.563;
   1:  PR[GP1:91,2] = PR[GP1:90,2] + 6.045;
   1:L PR[91] 10mm/sec CNT100;
   1:  PR[GP1:91,1] = PR[GP1:90,1] + 31.912;
   1:  PR[GP1:91,2] = PR[GP1:90,2] + 8.968;
   1:L PR[91] 10mm/sec CNT100;
   1:  PR[GP1:91,1] = PR[GP1:90,1] + 29.647;
   1:  PR[GP1:91,2] = PR[GP1:90,2] + 11.512;
   1:L PR[91] 10mm/sec CNT100;
   1:  PR[GP1:91,1] = PR[GP1:90,1] + 26.874;
   1:  PR[GP1:91,2] = PR[GP1:90,2] + 13.585;
   1:L PR[91] 10mm/sec CNT100;
   1:  PR[GP1:91,1] = PR[GP1:90,1] + 23.708;
   1:  PR[GP1:91,2] = PR[GP1:90,2] + 15.103;
   1:L PR[91] 10mm/sec CNT100;
   1:  PR[GP1:91,1] = PR[GP1:90,1] + 21.814;
   1:  PR[GP1:91,2] = PR[GP1:90,2] + 15.603;
   1:L PR[91] 10mm/sec CNT100;
   1:  PR[GP1:91,1] = PR[GP1:90,1] + 20.251;
   1:  PR[GP1:91,2] = PR[GP1:90,2] + 15.995;
   1:L PR[91] 10mm/sec CNT100;
   1:  PR[GP1:91,1] = PR[GP1:90,1] + 16.603;
   1:  PR[GP1:91,2] = PR[GP1:90,2] + 16.224;
   1:L PR[91] 10mm/sec CNT100;
   1:  PR[GP1:91,1] = PR[GP1:90,1] + 13.589;
   1:  PR[GP1:91,2] = PR[GP1:90,2] + 15.869;
   1:L PR[91] 10mm/sec CNT100;
   1:  PR[GP1:91,1] = PR[GP1:90,1] + 12.958;
   1:  PR[GP1:91,2] = PR[GP1:90,2] + 15.788;
   1:L PR[91] 10mm/sec CNT100;
   1:  PR[GP1:91,1] = PR[GP1:90,1] + 9.434;
   1:  PR[GP1:91,2] = PR[GP1:90,2] + 14.689;
   1:L PR[91] 10mm/sec CNT100;
   1:  PR[GP1:91,1] = PR[GP1:90,1] + 6.191;
   1:  PR[GP1:91,2] = PR[GP1:90,2] + 12.993;
   1:L PR[91] 10mm/sec CNT100;
   1:  PR[GP1:91,1] = PR[GP1:90,1] + 3.357;
   1:  PR[GP1:91,2] = PR[GP1:90,2] + 10.754;
   1:L PR[91] 10mm/sec CNT100;
   1:  PR[GP1:91,1] = PR[GP1:90,1] + 1.082;
   1:  PR[GP1:91,2] = PR[GP1:90,2] + 8.169;
   1:L PR[91] 10mm/sec CNT100;
   1:  PR[GP1:91,1] = PR[GP1:90,1] + 0.172;
   1:  PR[GP1:91,2] = PR[GP1:90,2] + 7.329;
   1:L PR[91] 10mm/sec CNT100;
   1:  PR[GP1:91,1] = PR[GP1:90,1] + -0.803;
   1:  PR[GP1:91,2] = PR[GP1:90,2] + 7.136;
   1:L PR[91] 10mm/sec CNT100;
   1:  PR[GP1:91,1] = PR[GP1:90,1] + -1.222;
   1:  PR[GP1:91,2] = PR[GP1:90,2] + 7.098;
   1:L PR[91] 10mm/sec CNT100;
   1:  PR[GP1:91,1] = PR[GP1:90,1] + -1.703;
   1:  PR[GP1:91,2] = PR[GP1:90,2] + 7.333;
   1:L PR[91] 10mm/sec CNT100;
   1:  PR[GP1:91,1] = PR[GP1:90,1] + -2.383;
   1:  PR[GP1:91,2] = PR[GP1:90,2] + 7.548;
   1:L PR[91] 10mm/sec CNT100;
   1:  PR[GP1:91,1] = PR[GP1:90,1] + -2.969;
   1:  PR[GP1:91,2] = PR[GP1:90,2] + 8.153;
   1:L PR[91] 10mm/sec CNT100;
   1:  PR[GP1:91,1] = PR[GP1:90,1] + -4.270;
   1:  PR[GP1:91,2] = PR[GP1:90,2] + 9.798;
   1:L PR[91] 10mm/sec CNT100;
   1:  PR[GP1:91,1] = PR[GP1:90,1] + -4.896;
   1:  PR[GP1:91,2] = PR[GP1:90,2] + 10.399;
   1:L PR[91] 10mm/sec CNT100;
   1:  PR[GP1:91,1] = PR[GP1:90,1] + -7.244;
   1:  PR[GP1:91,2] = PR[GP1:90,2] + 12.433;
   1:L PR[91] 10mm/sec CNT100;
   1:  PR[GP1:91,1] = PR[GP1:90,1] + -9.654;
   1:  PR[GP1:91,2] = PR[GP1:90,2] + 13.885;
   1:L PR[91] 10mm/sec CNT100;
   1:  PR[GP1:91,1] = PR[GP1:90,1] + -10.389;
   1:  PR[GP1:91,2] = PR[GP1:90,2] + 14.309;
   1:L PR[91] 10mm/sec CNT100;
   1:  PR[GP1:91,1] = PR[GP1:90,1] + -12.324;
   1:  PR[GP1:91,2] = PR[GP1:90,2] + 15.010;
   1:L PR[91] 10mm/sec CNT100;
   1:  PR[GP1:91,1] = PR[GP1:90,1] + -13.823;
   1:  PR[GP1:91,2] = PR[GP1:90,2] + 15.524;
   1:L PR[91] 10mm/sec CNT100;
   1:  PR[GP1:91,1] = PR[GP1:90,1] + -15.203;
   1:  PR[GP1:91,2] = PR[GP1:90,2] + 15.738;
   1:L PR[91] 10mm/sec CNT100;
   1:  PR[GP1:91,1] = PR[GP1:90,1] + -17.392;
   1:  PR[GP1:91,2] = PR[GP1:90,2] + 16.044;
   1:L PR[91] 10mm/sec CNT100;
   1:  PR[GP1:91,1] = PR[GP1:90,1] + -20.959;
   1:  PR[GP1:91,2] = PR[GP1:90,2] + 15.864;
   1:L PR[91] 10mm/sec CNT100;
   1:  PR[GP1:91,1] = PR[GP1:90,1] + -24.373;
   1:  PR[GP1:91,2] = PR[GP1:90,2] + 15.002;
   1:L PR[91] 10mm/sec CNT100;
   1:  PR[GP1:91,1] = PR[GP1:90,1] + -27.380;
   1:  PR[GP1:91,2] = PR[GP1:90,2] + 13.522;
   1:L PR[91] 10mm/sec CNT100;
   1:  PR[GP1:91,1] = PR[GP1:90,1] + -27.575;
   1:  PR[GP1:91,2] = PR[GP1:90,2] + 13.385;
   1:L PR[91] 10mm/sec CNT100;
   1:  PR[GP1:91,1] = PR[GP1:90,1] + -30.039;
   1:  PR[GP1:91,2] = PR[GP1:90,2] + 11.472;
   1:L PR[91] 10mm/sec CNT100;
   1:  PR[GP1:91,1] = PR[GP1:90,1] + -30.368;
   1:  PR[GP1:91,2] = PR[GP1:90,2] + 11.116;
   1:L PR[91] 10mm/sec CNT100;
   1:  PR[GP1:91,1] = PR[GP1:90,1] + -32.251;
   1:  PR[GP1:91,2] = PR[GP1:90,2] + 8.910;
   1:L PR[91] 10mm/sec CNT100;
   1:  PR[GP1:91,1] = PR[GP1:90,1] + -32.576;
   1:  PR[GP1:91,2] = PR[GP1:90,2] + 8.357;
   1:L PR[91] 10mm/sec CNT100;
   1:  PR[GP1:91,1] = PR[GP1:90,1] + -33.909;
   1:  PR[GP1:91,2] = PR[GP1:90,2] + 5.939;
   1:L PR[91] 10mm/sec CNT100;
   1:  PR[GP1:91,1] = PR[GP1:90,1] + -34.944;
   1:  PR[GP1:91,2] = PR[GP1:90,2] + 2.680;
   1:L PR[91] 10mm/sec CNT100;
   1:  PR[GP1:91,1] = PR[GP1:90,1] + -35.018;
   1:  PR[GP1:91,2] = PR[GP1:90,2] + 1.958;
   1:L PR[91] 10mm/sec CNT100;
   1:  PR[GP1:91,1] = PR[GP1:90,1] + -35.115;
   1:  PR[GP1:91,2] = PR[GP1:90,2] + 1.360;
   1:L PR[91] 10mm/sec CNT100;
   1:  PR[GP1:91,1] = PR[GP1:90,1] + -35.303;
   1:  PR[GP1:91,2] = PR[GP1:90,2] + -0.695;
   1:L PR[91] 10mm/sec CNT100;
   1:  PR[GP1:91,1] = PR[GP1:90,1] + -35.201;
   1:  PR[GP1:91,2] = PR[GP1:90,2] + -1.317;
   1:L PR[91] 10mm/sec CNT100;
   1:  PR[GP1:91,1] = PR[GP1:90,1] + -34.886;
   1:  PR[GP1:91,2] = PR[GP1:90,2] + -4.138;
   1:L PR[91] 10mm/sec CNT100;
   1:  PR[GP1:91,1] = PR[GP1:90,1] + -33.851;
   1:  PR[GP1:91,2] = PR[GP1:90,2] + -7.381;
   1:L PR[91] 10mm/sec CNT100;
   1:  PR[GP1:91,1] = PR[GP1:90,1] + -32.319;
   1:  PR[GP1:91,2] = PR[GP1:90,2] + -10.099;
   1:L PR[91] 10mm/sec CNT100;
   1:  PR[GP1:91,1] = PR[GP1:90,1] + -32.182;
   1:  PR[GP1:91,2] = PR[GP1:90,2] + -10.334;
   1:L PR[91] 10mm/sec CNT100;
   1:  PR[GP1:91,1] = PR[GP1:90,1] + -29.816;
   1:  PR[GP1:91,2] = PR[GP1:90,2] + -12.989;
   1:L PR[91] 10mm/sec CNT100;
   1:  PR[GP1:91,1] = PR[GP1:90,1] + -27.613;
   1:  PR[GP1:91,2] = PR[GP1:90,2] + -14.661;
   1:L PR[91] 10mm/sec CNT100;
   1:  PR[GP1:91,1] = PR[GP1:90,1] + -26.936;
   1:  PR[GP1:91,2] = PR[GP1:90,2] + -15.155;
   1:L PR[91] 10mm/sec CNT100;
   1:  PR[GP1:91,1] = PR[GP1:90,1] + -24.919;
   1:  PR[GP1:91,2] = PR[GP1:90,2] + -16.144;
   1:L PR[91] 10mm/sec CNT100;
   1:  PR[GP1:91,1] = PR[GP1:90,1] + -23.216;
   1:  PR[GP1:91,2] = PR[GP1:90,2] + -16.876;
   1:  PR[GP1:91,3] = PR[GP1:90,3] + 18.700;
   1:L PR[91] 10mm/sec CNT100;
   1:  PR[GP1:91,1] = PR[GP1:90,1] + -22.336;
   1:  PR[GP1:91,2] = PR[GP1:90,2] + -17.113;
   1:L PR[91] 10mm/sec CNT100;
   1:  PR[GP1:91,1] = PR[GP1:90,1] + -19.589;
   1:  PR[GP1:91,2] = PR[GP1:90,2] + -17.774;
   1:L PR[91] 10mm/sec CNT100;
   1:  PR[GP1:91,1] = PR[GP1:90,1] + -16.314;
   1:  PR[GP1:91,2] = PR[GP1:90,2] + -17.952;
   1:L PR[91] 10mm/sec CNT100;
   1:  PR[GP1:91,1] = PR[GP1:90,1] + -15.570;
   1:  PR[GP1:91,2] = PR[GP1:90,2] + -17.955;
   1:L PR[91] 10mm/sec CNT100;
   1:  PR[GP1:91,1] = PR[GP1:90,1] + -13.285;
   1:  PR[GP1:91,2] = PR[GP1:90,2] + -17.647;
   1:L PR[91] 10mm/sec CNT100;
   1:  PR[GP1:91,1] = PR[GP1:90,1] + -11.478;
   1:  PR[GP1:91,2] = PR[GP1:90,2] + -17.290;
   1:L PR[91] 10mm/sec CNT100;
   1:  PR[GP1:91,1] = PR[GP1:90,1] + -10.385;
   1:  PR[GP1:91,2] = PR[GP1:90,2] + -16.915;
   1:L PR[91] 10mm/sec CNT100;
   1:  PR[GP1:91,1] = PR[GP1:90,1] + -7.623;
   1:  PR[GP1:91,2] = PR[GP1:90,2] + -15.751;
   1:L PR[91] 10mm/sec CNT100;
   1:  PR[GP1:91,1] = PR[GP1:90,1] + -4.850;
   1:  PR[GP1:91,2] = PR[GP1:90,2] + -13.992;
   1:L PR[91] 10mm/sec CNT100;
   1:  PR[GP1:91,1] = PR[GP1:90,1] + -3.957;
   1:  PR[GP1:91,2] = PR[GP1:90,2] + -13.266;
   1:L PR[91] 10mm/sec CNT100;
   1:  PR[GP1:91,1] = PR[GP1:90,1] + -2.604;
   1:  PR[GP1:91,2] = PR[GP1:90,2] + -11.876;
   1:L PR[91] 10mm/sec CNT100;
   1:  PR[GP1:91,1] = PR[GP1:90,1] + -2.342;
   1:  PR[GP1:91,2] = PR[GP1:90,2] + -11.631;
   1:L PR[91] 10mm/sec CNT100;
   1:  PR[GP1:91,1] = PR[GP1:90,1] + -1.587;
   1:  PR[GP1:91,2] = PR[GP1:90,2] + -11.181;
   1:L PR[91] 10mm/sec CNT100;
   1:  PR[GP1:91,1] = PR[GP1:90,1] + -1.131;
   1:  PR[GP1:91,2] = PR[GP1:90,2] + -11.055;
   1:L PR[91] 10mm/sec CNT100;
   1:  PR[GP1:91,1] = PR[GP1:90,1] + -0.299;
   1:  PR[GP1:91,2] = PR[GP1:90,2] + -11.112;
   1:L PR[91] 10mm/sec CNT100;
   1:  PR[GP1:91,1] = PR[GP1:90,1] + 0.136;
   1:  PR[GP1:91,2] = PR[GP1:90,2] + -11.235;
   1:L PR[91] 10mm/sec CNT100;
   1:  PR[GP1:91,1] = PR[GP1:90,1] + 0.944;
   1:  PR[GP1:91,2] = PR[GP1:90,2] + -11.833;
   1:L PR[91] 10mm/sec CNT100;
   1:  PR[GP1:91,1] = PR[GP1:90,1] + 1.103;
   1:  PR[GP1:91,2] = PR[GP1:90,2] + -12.055;
   1:L PR[91] 10mm/sec CNT100;
   1:  PR[GP1:91,1] = PR[GP1:90,1] + 1.583;
   1:  PR[GP1:91,2] = PR[GP1:90,2] + -12.592;
   1:L PR[91] 10mm/sec CNT100;
   1:  PR[GP1:91,1] = PR[GP1:90,1] + 1.969;
   1:  PR[GP1:91,2] = PR[GP1:90,2] + -12.993;
   1:L PR[91] 10mm/sec CNT100;
   1:  PR[GP1:91,1] = PR[GP1:90,1] + 3.562;
   1:  PR[GP1:91,2] = PR[GP1:90,2] + -14.381;
   1:L PR[91] 10mm/sec CNT100;
   1:  PR[GP1:91,1] = PR[GP1:90,1] + 4.090;
   1:  PR[GP1:91,2] = PR[GP1:90,2] + -14.802;
   1:L PR[91] 10mm/sec CNT100;
   1:  PR[GP1:91,1] = PR[GP1:90,1] + 6.295;
   1:  PR[GP1:91,2] = PR[GP1:90,2] + -16.153;
   1:L PR[91] 10mm/sec CNT100;
   1:  PR[GP1:91,1] = PR[GP1:90,1] + 8.700;
   1:  PR[GP1:91,2] = PR[GP1:90,2] + -17.173;
   1:L PR[91] 10mm/sec CNT100;
   1:  PR[GP1:91,1] = PR[GP1:90,1] + 11.275;
   1:  PR[GP1:91,2] = PR[GP1:90,2] + -17.859;
   1:L PR[91] 10mm/sec CNT100;
   1:  PR[GP1:91,1] = PR[GP1:90,1] + 12.406;
   1:  PR[GP1:91,2] = PR[GP1:90,2] + -18.017;
   1:L PR[91] 10mm/sec CNT100;
   1:  PR[GP1:91,1] = PR[GP1:90,1] + 13.942;
   1:  PR[GP1:91,2] = PR[GP1:90,2] + -18.190;
   1:L PR[91] 10mm/sec CNT100;
   1:  PR[GP1:91,1] = PR[GP1:90,1] + 16.171;
   1:  PR[GP1:91,2] = PR[GP1:90,2] + -18.174;
   1:L PR[91] 10mm/sec CNT100;
   1:  PR[GP1:91,1] = PR[GP1:90,1] + 16.667;
   1:  PR[GP1:91,2] = PR[GP1:90,2] + -18.159;
   1:L PR[91] 10mm/sec CNT100;
   1:  PR[GP1:91,1] = PR[GP1:90,1] + 17.924;
   1:  PR[GP1:91,2] = PR[GP1:90,2] + -17.969;
   1:L PR[91] 10mm/sec CNT100;
   1:  PR[GP1:91,1] = PR[GP1:90,1] + 19.435;
   1:  PR[GP1:91,2] = PR[GP1:90,2] + -17.768;
   1:L PR[91] 10mm/sec CNT100;
   1:  PR[GP1:91,1] = PR[GP1:90,1] + 22.149;
   1:  PR[GP1:91,2] = PR[GP1:90,2] + -17.016;
   1:L PR[91] 10mm/sec CNT100;
   1:  PR[GP1:91,1] = PR[GP1:90,1] + 24.169;
   1:  PR[GP1:91,2] = PR[GP1:90,2] + -16.156;
   1:L PR[91] 10mm/sec CNT100;
   1:  PR[GP1:91,1] = PR[GP1:90,1] + 24.746;
   1:  PR[GP1:91,2] = PR[GP1:90,2] + -15.901;
   1:L PR[91] 10mm/sec CNT100;
   1:  PR[GP1:91,1] = PR[GP1:90,1] + 27.179;
   1:  PR[GP1:91,2] = PR[GP1:90,2] + -14.419;
   1:L PR[91] 10mm/sec CNT100;
   1:  PR[GP1:91,1] = PR[GP1:90,1] + 29.347;
   1:  PR[GP1:91,2] = PR[GP1:90,2] + -12.608;
   1:L PR[91] 10mm/sec CNT100;
   1:  PR[GP1:91,1] = PR[GP1:90,1] + 31.189;
   1:  PR[GP1:91,2] = PR[GP1:90,2] + -10.520;
   1:L PR[91] 10mm/sec CNT100;
   1:  PR[GP1:91,1] = PR[GP1:90,1] + 32.665;
   1:  PR[GP1:91,2] = PR[GP1:90,2] + -8.207;
   1:L PR[91] 10mm/sec CNT100;
   1:  PR[GP1:91,1] = PR[GP1:90,1] + 33.745;
   1:  PR[GP1:91,2] = PR[GP1:90,2] + -5.726;
   1:L PR[91] 10mm/sec CNT100;
   1:  PR[GP1:91,1] = PR[GP1:90,1] + 34.396;
   1:  PR[GP1:91,2] = PR[GP1:90,2] + -3.137;
   1:L PR[91] 10mm/sec CNT100;
   1:  PR[GP1:91,1] = PR[GP1:90,1] + 34.603;
   1:  PR[GP1:91,2] = PR[GP1:90,2] + -0.504;
   1:L PR[91] 10mm/sec CNT100;
   1:  PR[GP1:91,1] = PR[GP1:90,1] + 34.237;
   1:  PR[GP1:91,2] = PR[GP1:90,2] + 2.823;
   1:L PR[91] 10mm/sec CNT100;
   1:  PR[GP1:91,1] = PR[GP1:90,1] + 33.202;
   1:  PR[GP1:91,2] = PR[GP1:90,2] + 6.007;
   1:L PR[91] 10mm/sec CNT100;
   1:  PR[GP1:91,1] = PR[GP1:90,1] + 31.513;
   1:  PR[GP1:91,2] = PR[GP1:90,2] + 8.927;
   1:L PR[91] 10mm/sec CNT100;
   1:  PR[GP1:91,1] = PR[GP1:90,1] + 29.235;
   1:  PR[GP1:91,2] = PR[GP1:90,2] + 11.473;
   1:L PR[91] 10mm/sec CNT100;
   1:  PR[GP1:91,1] = PR[GP1:90,1] + 26.458;
   1:  PR[GP1:91,2] = PR[GP1:90,2] + 13.545;
   1:L PR[91] 10mm/sec CNT100;
   1:  PR[GP1:91,1] = PR[GP1:90,1] + 23.902;
   1:  PR[GP1:91,2] = PR[GP1:90,2] + 14.769;
   1:L PR[91] 10mm/sec CNT100;
   1:  PR[GP1:91,1] = PR[GP1:90,1] + 23.284;
   1:  PR[GP1:91,2] = PR[GP1:90,2] + 15.054;
   1:L PR[91] 10mm/sec CNT100;
   1:  PR[GP1:91,1] = PR[GP1:90,1] + 19.770;
   1:  PR[GP1:91,2] = PR[GP1:90,2] + 15.934;
   1:L PR[91] 10mm/sec CNT100;
   1:  PR[GP1:91,1] = PR[GP1:90,1] + 16.113;
   1:  PR[GP1:91,2] = PR[GP1:90,2] + 16.157;
   1:L PR[91] 10mm/sec CNT100;
   1:  PR[GP1:91,1] = PR[GP1:90,1] + 14.954;
   1:  PR[GP1:91,2] = PR[GP1:90,2] + 16.021;
   1:L PR[91] 10mm/sec CNT100;
   1:  PR[GP1:91,1] = PR[GP1:90,1] + 12.460;
   1:  PR[GP1:91,2] = PR[GP1:90,2] + 15.703;
   1:L PR[91] 10mm/sec CNT100;
   1:  PR[GP1:91,1] = PR[GP1:90,1] + 8.934;
   1:  PR[GP1:91,2] = PR[GP1:90,2] + 14.603;
   1:L PR[91] 10mm/sec CNT100;
   1:  PR[GP1:91,1] = PR[GP1:90,1] + 7.920;
   1:  PR[GP1:91,2] = PR[GP1:90,2] + 14.077;
   1:L PR[91] 10mm/sec CNT100;
   1:  PR[GP1:91,1] = PR[GP1:90,1] + 5.712;
   1:  PR[GP1:91,2] = PR[GP1:90,2] + 12.896;
   1:L PR[91] 10mm/sec CNT100;
   1:  PR[GP1:91,1] = PR[GP1:90,1] + 2.861;
   1:  PR[GP1:91,2] = PR[GP1:90,2] + 10.657;
   1:L PR[91] 10mm/sec CNT100;
   1:  PR[GP1:91,1] = PR[GP1:90,1] + 1.040;
   1:  PR[GP1:91,2] = PR[GP1:90,2] + 8.645;
   1:L PR[91] 10mm/sec CNT100;
   1:  PR[GP1:91,1] = PR[GP1:90,1] + 0.123;
   1:  PR[GP1:91,2] = PR[GP1:90,2] + 7.819;
   1:L PR[91] 10mm/sec CNT100;
   1:  PR[GP1:91,1] = PR[GP1:90,1] + -0.584;
   1:  PR[GP1:91,2] = PR[GP1:90,2] + 7.679;
   1:L PR[91] 10mm/sec CNT100;
   1:  PR[GP1:91,1] = PR[GP1:90,1] + -1.270;
   1:  PR[GP1:91,2] = PR[GP1:90,2] + 7.616;
   1:L PR[91] 10mm/sec CNT100;
   1:  PR[GP1:91,1] = PR[GP1:90,1] + -2.224;
   1:  PR[GP1:91,2] = PR[GP1:90,2] + 8.082;
   1:L PR[91] 10mm/sec CNT100;
   1:  PR[GP1:91,1] = PR[GP1:90,1] + -2.441;
   1:  PR[GP1:91,2] = PR[GP1:90,2] + 8.151;
   1:L PR[91] 10mm/sec CNT100;
   1:  PR[GP1:91,1] = PR[GP1:90,1] + -2.923;
   1:  PR[GP1:91,2] = PR[GP1:90,2] + 8.628;
   1:L PR[91] 10mm/sec CNT100;
   1:  PR[GP1:91,1] = PR[GP1:90,1] + -3.578;
   1:  PR[GP1:91,2] = PR[GP1:90,2] + 9.445;
   1:L PR[91] 10mm/sec CNT100;
   1:  PR[GP1:91,1] = PR[GP1:90,1] + -4.926;
   1:  PR[GP1:91,2] = PR[GP1:90,2] + 10.738;
   1:L PR[91] 10mm/sec CNT100;
   1:  PR[GP1:91,1] = PR[GP1:90,1] + -6.607;
   1:  PR[GP1:91,2] = PR[GP1:90,2] + 12.187;
   1:L PR[91] 10mm/sec CNT100;
   1:  PR[GP1:91,1] = PR[GP1:90,1] + -7.230;
   1:  PR[GP1:91,2] = PR[GP1:90,2] + 12.584;
   1:L PR[91] 10mm/sec CNT100;
   1:  PR[GP1:91,1] = PR[GP1:90,1] + -9.988;
   1:  PR[GP1:91,2] = PR[GP1:90,2] + 14.186;
   1:L PR[91] 10mm/sec CNT100;
   1:  PR[GP1:91,1] = PR[GP1:90,1] + -12.596;
   1:  PR[GP1:91,2] = PR[GP1:90,2] + 15.131;
   1:L PR[91] 10mm/sec CNT100;
   1:  PR[GP1:91,1] = PR[GP1:90,1] + -13.431;
   1:  PR[GP1:91,2] = PR[GP1:90,2] + 15.418;
   1:L PR[91] 10mm/sec CNT100;
   1:  PR[GP1:91,1] = PR[GP1:90,1] + -15.470;
   1:  PR[GP1:91,2] = PR[GP1:90,2] + 15.734;
   1:L PR[91] 10mm/sec CNT100;
   1:  PR[GP1:91,1] = PR[GP1:90,1] + -17.016;
   1:  PR[GP1:91,2] = PR[GP1:90,2] + 15.950;
   1:L PR[91] 10mm/sec CNT100;
   1:  PR[GP1:91,1] = PR[GP1:90,1] + -18.471;
   1:  PR[GP1:91,2] = PR[GP1:90,2] + 15.890;
   1:L PR[91] 10mm/sec CNT100;
   1:  PR[GP1:91,1] = PR[GP1:90,1] + -20.591;
   1:  PR[GP1:91,2] = PR[GP1:90,2] + 15.776;
   1:L PR[91] 10mm/sec CNT100;
   1:  PR[GP1:91,1] = PR[GP1:90,1] + -24.023;
   1:  PR[GP1:91,2] = PR[GP1:90,2] + 14.916;
   1:L PR[91] 10mm/sec CNT100;
   1:  PR[GP1:91,1] = PR[GP1:90,1] + -24.509;
   1:  PR[GP1:91,2] = PR[GP1:90,2] + 14.688;
   1:L PR[91] 10mm/sec CNT100;
   1:  PR[GP1:91,1] = PR[GP1:90,1] + -27.169;
   1:  PR[GP1:91,2] = PR[GP1:90,2] + 13.415;
   1:L PR[91] 10mm/sec CNT100;
   1:  PR[GP1:91,1] = PR[GP1:90,1] + -29.913;
   1:  PR[GP1:91,2] = PR[GP1:90,2] + 11.341;
   1:L PR[91] 10mm/sec CNT100;
   1:  PR[GP1:91,1] = PR[GP1:90,1] + -32.105;
   1:  PR[GP1:91,2] = PR[GP1:90,2] + 8.785;
   1:L PR[91] 10mm/sec CNT100;
   1:  PR[GP1:91,1] = PR[GP1:90,1] + -33.740;
   1:  PR[GP1:91,2] = PR[GP1:90,2] + 5.825;
   1:L PR[91] 10mm/sec CNT100;
   1:  PR[GP1:91,1] = PR[GP1:90,1] + -34.762;
   1:  PR[GP1:91,2] = PR[GP1:90,2] + 2.583;
   1:L PR[91] 10mm/sec CNT100;
   1:  PR[GP1:91,1] = PR[GP1:90,1] + -34.803;
   1:  PR[GP1:91,2] = PR[GP1:90,2] + 2.264;
   1:L PR[91] 10mm/sec CNT100;
   1:  PR[GP1:91,1] = PR[GP1:90,1] + -35.082;
   1:  PR[GP1:91,2] = PR[GP1:90,2] + -0.785;
   1:L PR[91] 10mm/sec CNT100;
   1:  PR[GP1:91,1] = PR[GP1:90,1] + -34.689;
   1:  PR[GP1:91,2] = PR[GP1:90,2] + -4.175;
   1:L PR[91] 10mm/sec CNT100;
   1:  PR[GP1:91,1] = PR[GP1:90,1] + -33.602;
   1:  PR[GP1:91,2] = PR[GP1:90,2] + -7.442;
   1:L PR[91] 10mm/sec CNT100;
   1:  PR[GP1:91,1] = PR[GP1:90,1] + -32.109;
   1:  PR[GP1:91,2] = PR[GP1:90,2] + -10.008;
   1:L PR[91] 10mm/sec CNT100;
   1:  PR[GP1:91,1] = PR[GP1:90,1] + -31.834;
   1:  PR[GP1:91,2] = PR[GP1:90,2] + -10.468;
   1:L PR[91] 10mm/sec CNT100;
   1:  PR[GP1:91,1] = PR[GP1:90,1] + -30.098;
   1:  PR[GP1:91,2] = PR[GP1:90,2] + -12.424;
   1:L PR[91] 10mm/sec CNT100;
   1:  PR[GP1:91,1] = PR[GP1:90,1] + -29.452;
   1:  PR[GP1:91,2] = PR[GP1:90,2] + -13.128;
   1:L PR[91] 10mm/sec CNT100;
   1:  PR[GP1:91,1] = PR[GP1:90,1] + -27.733;
   1:  PR[GP1:91,2] = PR[GP1:90,2] + -14.433;
   1:L PR[91] 10mm/sec CNT100;
   1:  PR[GP1:91,1] = PR[GP1:90,1] + -26.546;
   1:  PR[GP1:91,2] = PR[GP1:90,2] + -15.298;
   1:L PR[91] 10mm/sec CNT100;
   1:  PR[GP1:91,1] = PR[GP1:90,1] + -25.116;
   1:  PR[GP1:91,2] = PR[GP1:90,2] + -15.999;
   1:L PR[91] 10mm/sec CNT100;
   1:  PR[GP1:91,1] = PR[GP1:90,1] + -22.805;
   1:  PR[GP1:91,2] = PR[GP1:90,2] + -17.013;
   1:  PR[GP1:91,3] = PR[GP1:90,3] + 19.800;
   1:L PR[91] 10mm/sec CNT100;
   1:  PR[GP1:91,1] = PR[GP1:90,1] + -19.523;
   1:  PR[GP1:91,2] = PR[GP1:90,2] + -17.828;
   1:L PR[91] 10mm/sec CNT100;
   1:  PR[GP1:91,1] = PR[GP1:90,1] + -18.962;
   1:  PR[GP1:91,2] = PR[GP1:90,2] + -17.941;
   1:L PR[91] 10mm/sec CNT100;
   1:  PR[GP1:91,1] = PR[GP1:90,1] + -16.458;
   1:  PR[GP1:91,2] = PR[GP1:90,2] + -18.084;
   1:L PR[91] 10mm/sec CNT100;
   1:  PR[GP1:91,1] = PR[GP1:90,1] + -14.819;
   1:  PR[GP1:91,2] = PR[GP1:90,2] + -18.090;
   1:L PR[91] 10mm/sec CNT100;
   1:  PR[GP1:91,1] = PR[GP1:90,1] + -13.450;
   1:  PR[GP1:91,2] = PR[GP1:90,2] + -17.906;
   1:L PR[91] 10mm/sec CNT100;
   1:  PR[GP1:91,1] = PR[GP1:90,1] + -10.677;
   1:  PR[GP1:91,2] = PR[GP1:90,2] + -17.359;
   1:L PR[91] 10mm/sec CNT100;
   1:  PR[GP1:91,1] = PR[GP1:90,1] + -10.545;
   1:  PR[GP1:91,2] = PR[GP1:90,2] + -17.313;
   1:L PR[91] 10mm/sec CNT100;
   1:  PR[GP1:91,1] = PR[GP1:90,1] + -10.056;
   1:  PR[GP1:91,2] = PR[GP1:90,2] + -17.107;
   1:L PR[91] 10mm/sec CNT100;
   1:  PR[GP1:91,1] = PR[GP1:90,1] + -7.412;
   1:  PR[GP1:91,2] = PR[GP1:90,2] + -16.134;
   1:L PR[91] 10mm/sec CNT100;
   1:  PR[GP1:91,1] = PR[GP1:90,1] + -6.358;
   1:  PR[GP1:91,2] = PR[GP1:90,2] + -15.598;
   1:L PR[91] 10mm/sec CNT100;
   1:  PR[GP1:91,1] = PR[GP1:90,1] + -4.717;
   1:  PR[GP1:91,2] = PR[GP1:90,2] + -14.560;
   1:L PR[91] 10mm/sec CNT100;
   1:  PR[GP1:91,1] = PR[GP1:90,1] + -2.772;
   1:  PR[GP1:91,2] = PR[GP1:90,2] + -12.979;
   1:L PR[91] 10mm/sec CNT100;
   1:  PR[GP1:91,1] = PR[GP1:90,1] + -2.368;
   1:  PR[GP1:91,2] = PR[GP1:90,2] + -12.561;
   1:L PR[91] 10mm/sec CNT100;
   1:  PR[GP1:91,1] = PR[GP1:90,1] + -1.267;
   1:  PR[GP1:91,2] = PR[GP1:90,2] + -11.932;
   1:L PR[91] 10mm/sec CNT100;
   1:  PR[GP1:91,1] = PR[GP1:90,1] + 0.040;
   1:  PR[GP1:91,2] = PR[GP1:90,2] + -12.023;
   1:L PR[91] 10mm/sec CNT100;
   1:  PR[GP1:91,1] = PR[GP1:90,1] + 1.080;
   1:  PR[GP1:91,2] = PR[GP1:90,2] + -12.725;
   1:L PR[91] 10mm/sec CNT100;
   1:  PR[GP1:91,1] = PR[GP1:90,1] + 1.546;
   1:  PR[GP1:91,2] = PR[GP1:90,2] + -13.210;
   1:L PR[91] 10mm/sec CNT100;
   1:  PR[GP1:91,1] = PR[GP1:90,1] + 2.703;
   1:  PR[GP1:91,2] = PR[GP1:90,2] + -14.227;
   1:L PR[91] 10mm/sec CNT100;
   1:  PR[GP1:91,1] = PR[GP1:90,1] + 3.798;
   1:  PR[GP1:91,2] = PR[GP1:90,2] + -15.100;
   1:L PR[91] 10mm/sec CNT100;
   1:  PR[GP1:91,1] = PR[GP1:90,1] + 5.116;
   1:  PR[GP1:91,2] = PR[GP1:90,2] + -15.915;
   1:L PR[91] 10mm/sec CNT100;
   1:  PR[GP1:91,1] = PR[GP1:90,1] + 6.003;
   1:  PR[GP1:91,2] = PR[GP1:90,2] + -16.421;
   1:L PR[91] 10mm/sec CNT100;
   1:  PR[GP1:91,1] = PR[GP1:90,1] + 7.921;
   1:  PR[GP1:91,2] = PR[GP1:90,2] + -17.226;
   1:L PR[91] 10mm/sec CNT100;
   1:  PR[GP1:91,1] = PR[GP1:90,1] + 8.405;
   1:  PR[GP1:91,2] = PR[GP1:90,2] + -17.412;
   1:L PR[91] 10mm/sec CNT100;
   1:  PR[GP1:91,1] = PR[GP1:90,1] + 10.970;
   1:  PR[GP1:91,2] = PR[GP1:90,2] + -18.059;
   1:L PR[91] 10mm/sec CNT100;
   1:  PR[GP1:91,1] = PR[GP1:90,1] + 13.649;
   1:  PR[GP1:91,2] = PR[GP1:90,2] + -18.364;
   1:L PR[91] 10mm/sec CNT100;
   1:  PR[GP1:91,1] = PR[GP1:90,1] + 14.755;
   1:  PR[GP1:91,2] = PR[GP1:90,2] + -18.356;
   1:L PR[91] 10mm/sec CNT100;
   1:  PR[GP1:91,1] = PR[GP1:90,1] + 16.366;
   1:  PR[GP1:91,2] = PR[GP1:90,2] + -18.307;
   1:L PR[91] 10mm/sec CNT100;
   1:  PR[GP1:91,1] = PR[GP1:90,1] + 19.091;
   1:  PR[GP1:91,2] = PR[GP1:90,2] + -17.885;
   1:L PR[91] 10mm/sec CNT100;
   1:  PR[GP1:91,1] = PR[GP1:90,1] + 20.138;
   1:  PR[GP1:91,2] = PR[GP1:90,2] + -17.570;
   1:L PR[91] 10mm/sec CNT100;
   1:  PR[GP1:91,1] = PR[GP1:90,1] + 21.788;
   1:  PR[GP1:91,2] = PR[GP1:90,2] + -17.105;
   1:L PR[91] 10mm/sec CNT100;
   1:  PR[GP1:91,1] = PR[GP1:90,1] + 24.374;
   1:  PR[GP1:91,2] = PR[GP1:90,2] + -15.974;
   1:L PR[91] 10mm/sec CNT100;
   1:  PR[GP1:91,1] = PR[GP1:90,1] + 26.215;
   1:  PR[GP1:91,2] = PR[GP1:90,2] + -14.852;
   1:L PR[91] 10mm/sec CNT100;
   1:  PR[GP1:91,1] = PR[GP1:90,1] + 26.779;
   1:  PR[GP1:91,2] = PR[GP1:90,2] + -14.499;
   1:L PR[91] 10mm/sec CNT100;
   1:  PR[GP1:91,1] = PR[GP1:90,1] + 28.945;
   1:  PR[GP1:91,2] = PR[GP1:90,2] + -12.691;
   1:L PR[91] 10mm/sec CNT100;
   1:  PR[GP1:91,1] = PR[GP1:90,1] + 30.788;
   1:  PR[GP1:91,2] = PR[GP1:90,2] + -10.596;
   1:L PR[91] 10mm/sec CNT100;
   1:  PR[GP1:91,1] = PR[GP1:90,1] + 32.264;
   1:  PR[GP1:91,2] = PR[GP1:90,2] + -8.276;
   1:L PR[91] 10mm/sec CNT100;
   1:  PR[GP1:91,1] = PR[GP1:90,1] + 33.343;
   1:  PR[GP1:91,2] = PR[GP1:90,2] + -5.788;
   1:L PR[91] 10mm/sec CNT100;
   1:  PR[GP1:91,1] = PR[GP1:90,1] + 33.999;
   1:  PR[GP1:91,2] = PR[GP1:90,2] + -3.189;
   1:L PR[91] 10mm/sec CNT100;
   1:  PR[GP1:91,1] = PR[GP1:90,1] + 34.177;
   1:  PR[GP1:91,2] = PR[GP1:90,2] + -1.041;
   1:L PR[91] 10mm/sec CNT100;
   1:  PR[GP1:91,1] = PR[GP1:90,1] + 34.232;
   1:  PR[GP1:91,2] = PR[GP1:90,2] + -0.537;
   1:L PR[91] 10mm/sec CNT100;
   1:  PR[GP1:91,1] = PR[GP1:90,1] + 33.843;
   1:  PR[GP1:91,2] = PR[GP1:90,2] + 2.779;
   1:L PR[91] 10mm/sec CNT100;
   1:  PR[GP1:91,1] = PR[GP1:90,1] + 32.800;
   1:  PR[GP1:91,2] = PR[GP1:90,2] + 5.966;
   1:L PR[91] 10mm/sec CNT100;
   1:  PR[GP1:91,1] = PR[GP1:90,1] + 31.105;
   1:  PR[GP1:91,2] = PR[GP1:90,2] + 8.888;
   1:L PR[91] 10mm/sec CNT100;
   1:  PR[GP1:91,1] = PR[GP1:90,1] + 28.823;
   1:  PR[GP1:91,2] = PR[GP1:90,2] + 11.434;
   1:L PR[91] 10mm/sec CNT100;
   1:  PR[GP1:91,1] = PR[GP1:90,1] + 26.038;
   1:  PR[GP1:91,2] = PR[GP1:90,2] + 13.500;
   1:L PR[91] 10mm/sec CNT100;
   1:  PR[GP1:91,1] = PR[GP1:90,1] + 22.801;
   1:  PR[GP1:91,2] = PR[GP1:90,2] + 14.993;
   1:L PR[91] 10mm/sec CNT100;
   1:  PR[GP1:91,1] = PR[GP1:90,1] + 19.291;
   1:  PR[GP1:91,2] = PR[GP1:90,2] + 15.874;
   1:L PR[91] 10mm/sec CNT100;
   1:  PR[GP1:91,1] = PR[GP1:90,1] + 15.626;
   1:  PR[GP1:91,2] = PR[GP1:90,2] + 16.082;
   1:L PR[91] 10mm/sec CNT100;
   1:  PR[GP1:91,1] = PR[GP1:90,1] + 14.684;
   1:  PR[GP1:91,2] = PR[GP1:90,2] + 15.964;
   1:L PR[91] 10mm/sec CNT100;
   1:  PR[GP1:91,1] = PR[GP1:90,1] + 11.963;
   1:  PR[GP1:91,2] = PR[GP1:90,2] + 15.617;
   1:L PR[91] 10mm/sec CNT100;
   1:  PR[GP1:91,1] = PR[GP1:90,1] + 8.449;
   1:  PR[GP1:91,2] = PR[GP1:90,2] + 14.513;
   1:L PR[91] 10mm/sec CNT100;
   1:  PR[GP1:91,1] = PR[GP1:90,1] + 5.231;
   1:  PR[GP1:91,2] = PR[GP1:90,2] + 12.797;
   1:L PR[91] 10mm/sec CNT100;
   1:  PR[GP1:91,1] = PR[GP1:90,1] + 3.619;
   1:  PR[GP1:91,2] = PR[GP1:90,2] + 11.532;
   1:L PR[91] 10mm/sec CNT100;
   1:  PR[GP1:91,1] = PR[GP1:90,1] + 2.409;
   1:  PR[GP1:91,2] = PR[GP1:90,2] + 10.550;
   1:L PR[91] 10mm/sec CNT100;
   1:  PR[GP1:91,1] = PR[GP1:90,1] + 0.995;
   1:  PR[GP1:91,2] = PR[GP1:90,2] + 8.996;
   1:L PR[91] 10mm/sec CNT100;
   1:  PR[GP1:91,1] = PR[GP1:90,1] + 0.556;
   1:  PR[GP1:91,2] = PR[GP1:90,2] + 8.739;
   1:L PR[91] 10mm/sec CNT100;
   1:  PR[GP1:91,1] = PR[GP1:90,1] + 0.078;
   1:  PR[GP1:91,2] = PR[GP1:90,2] + 8.310;
   1:L PR[91] 10mm/sec CNT100;
   1:  PR[GP1:91,1] = PR[GP1:90,1] + -0.366;
   1:  PR[GP1:91,2] = PR[GP1:90,2] + 8.222;
   1:L PR[91] 10mm/sec CNT100;
   1:  PR[GP1:91,1] = PR[GP1:90,1] + -1.318;
   1:  PR[GP1:91,2] = PR[GP1:90,2] + 8.135;
   1:L PR[91] 10mm/sec CNT100;
   1:  PR[GP1:91,1] = PR[GP1:90,1] + -1.994;
   1:  PR[GP1:91,2] = PR[GP1:90,2] + 8.465;
   1:L PR[91] 10mm/sec CNT100;
   1:  PR[GP1:91,1] = PR[GP1:90,1] + -2.492;
   1:  PR[GP1:91,2] = PR[GP1:90,2] + 8.681;
   1:L PR[91] 10mm/sec CNT100;
   1:  PR[GP1:91,1] = PR[GP1:90,1] + -2.867;
   1:  PR[GP1:91,2] = PR[GP1:90,2] + 9.074;
   1:L PR[91] 10mm/sec CNT100;
   1:  PR[GP1:91,1] = PR[GP1:90,1] + -4.957;
   1:  PR[GP1:91,2] = PR[GP1:90,2] + 11.077;
   1:L PR[91] 10mm/sec CNT100;
   1:  PR[GP1:91,1] = PR[GP1:90,1] + -5.940;
   1:  PR[GP1:91,2] = PR[GP1:90,2] + 11.925;
   1:L PR[91] 10mm/sec CNT100;
   1:  PR[GP1:91,1] = PR[GP1:90,1] + -7.309;
   1:  PR[GP1:91,2] = PR[GP1:90,2] + 12.797;
   1:L PR[91] 10mm/sec CNT100;
   1:  PR[GP1:91,1] = PR[GP1:90,1] + -9.396;
   1:  PR[GP1:91,2] = PR[GP1:90,2] + 14.001;
   1:L PR[91] 10mm/sec CNT100;
   1:  PR[GP1:91,1] = PR[GP1:90,1] + -9.940;
   1:  PR[GP1:91,2] = PR[GP1:90,2] + 14.215;
   1:L PR[91] 10mm/sec CNT100;
   1:  PR[GP1:91,1] = PR[GP1:90,1] + -13.043;
   1:  PR[GP1:91,2] = PR[GP1:90,2] + 15.312;
   1:L PR[91] 10mm/sec CNT100;
   1:  PR[GP1:91,1] = PR[GP1:90,1] + -15.738;
   1:  PR[GP1:91,2] = PR[GP1:90,2] + 15.729;
   1:L PR[91] 10mm/sec CNT100;
   1:  PR[GP1:91,1] = PR[GP1:90,1] + -16.637;
   1:  PR[GP1:91,2] = PR[GP1:90,2] + 15.855;
   1:L PR[91] 10mm/sec CNT100;
   1:  PR[GP1:91,1] = PR[GP1:90,1] + -18.717;
   1:  PR[GP1:91,2] = PR[GP1:90,2] + 15.770;
   1:L PR[91] 10mm/sec CNT100;
   1:  PR[GP1:91,1] = PR[GP1:90,1] + -20.225;
   1:  PR[GP1:91,2] = PR[GP1:90,2] + 15.689;
   1:L PR[91] 10mm/sec CNT100;
   1:  PR[GP1:91,1] = PR[GP1:90,1] + -23.666;
   1:  PR[GP1:91,2] = PR[GP1:90,2] + 14.832;
   1:L PR[91] 10mm/sec CNT100;
   1:  PR[GP1:91,1] = PR[GP1:90,1] + -26.825;
   1:  PR[GP1:91,2] = PR[GP1:90,2] + 13.330;
   1:L PR[91] 10mm/sec CNT100;
   1:  PR[GP1:91,1] = PR[GP1:90,1] + -27.437;
   1:  PR[GP1:91,2] = PR[GP1:90,2] + 12.874;
   1:L PR[91] 10mm/sec CNT100;
   1:  PR[GP1:91,1] = PR[GP1:90,1] + -29.578;
   1:  PR[GP1:91,2] = PR[GP1:90,2] + 11.253;
   1:L PR[91] 10mm/sec CNT100;
   1:  PR[GP1:91,1] = PR[GP1:90,1] + -31.820;
   1:  PR[GP1:91,2] = PR[GP1:90,2] + 8.681;
   1:L PR[91] 10mm/sec CNT100;
   1:  PR[GP1:91,1] = PR[GP1:90,1] + -33.475;
   1:  PR[GP1:91,2] = PR[GP1:90,2] + 5.721;
   1:L PR[91] 10mm/sec CNT100;
   1:  PR[GP1:91,1] = PR[GP1:90,1] + -34.490;
   1:  PR[GP1:91,2] = PR[GP1:90,2] + 2.500;
   1:L PR[91] 10mm/sec CNT100;
   1:  PR[GP1:91,1] = PR[GP1:90,1] + -34.783;
   1:  PR[GP1:91,2] = PR[GP1:90,2] + -0.880;
   1:L PR[91] 10mm/sec CNT100;
   1:  PR[GP1:91,1] = PR[GP1:90,1] + -34.359;
   1:  PR[GP1:91,2] = PR[GP1:90,2] + -4.292;
   1:L PR[91] 10mm/sec CNT100;
   1:  PR[GP1:91,1] = PR[GP1:90,1] + -33.265;
   1:  PR[GP1:91,2] = PR[GP1:90,2] + -7.570;
   1:L PR[91] 10mm/sec CNT100;
   1:  PR[GP1:91,1] = PR[GP1:90,1] + -32.053;
   1:  PR[GP1:91,2] = PR[GP1:90,2] + -9.654;
   1:L PR[91] 10mm/sec CNT100;
   1:  PR[GP1:91,1] = PR[GP1:90,1] + -31.484;
   1:  PR[GP1:91,2] = PR[GP1:90,2] + -10.605;
   1:L PR[91] 10mm/sec CNT100;
   1:  PR[GP1:91,1] = PR[GP1:90,1] + -30.133;
   1:  PR[GP1:91,2] = PR[GP1:90,2] + -12.126;
   1:L PR[91] 10mm/sec CNT100;
   1:  PR[GP1:91,1] = PR[GP1:90,1] + -29.084;
   1:  PR[GP1:91,2] = PR[GP1:90,2] + -13.271;
   1:L PR[91] 10mm/sec CNT100;
   1:  PR[GP1:91,1] = PR[GP1:90,1] + -27.854;
   1:  PR[GP1:91,2] = PR[GP1:90,2] + -14.205;
   1:L PR[91] 10mm/sec CNT100;
   1:  PR[GP1:91,1] = PR[GP1:90,1] + -26.156;
   1:  PR[GP1:91,2] = PR[GP1:90,2] + -15.442;
   1:L PR[91] 10mm/sec CNT100;
   1:  PR[GP1:91,1] = PR[GP1:90,1] + -25.313;
   1:  PR[GP1:91,2] = PR[GP1:90,2] + -15.855;
   1:L PR[91] 10mm/sec CNT100;
   1:  PR[GP1:91,1] = PR[GP1:90,1] + -22.632;
   1:  PR[GP1:91,2] = PR[GP1:90,2] + -17.037;
   1:  PR[GP1:91,3] = PR[GP1:90,3] + 20.900;
   1:L PR[91] 10mm/sec CNT100;
   1:  PR[GP1:91,1] = PR[GP1:90,1] + -22.265;
   1:  PR[GP1:91,2] = PR[GP1:90,2] + -17.189;
   1:L PR[91] 10mm/sec CNT100;
   1:  PR[GP1:91,1] = PR[GP1:90,1] + -19.630;
   1:  PR[GP1:91,2] = PR[GP1:90,2] + -17.847;
   1:L PR[91] 10mm/sec CNT100;
   1:  PR[GP1:91,1] = PR[GP1:90,1] + -18.269;
   1:  PR[GP1:91,2] = PR[GP1:90,2] + -18.121;
   1:L PR[91] 10mm/sec CNT100;
   1:  PR[GP1:91,1] = PR[GP1:90,1] + -16.603;
   1:  PR[GP1:91,2] = PR[GP1:90,2] + -18.216;
   1:L PR[91] 10mm/sec CNT100;
   1:  PR[GP1:91,1] = PR[GP1:90,1] + -14.069;
   1:  PR[GP1:91,2] = PR[GP1:90,2] + -18.226;
   1:L PR[91] 10mm/sec CNT100;
   1:  PR[GP1:91,1] = PR[GP1:90,1] + -13.615;
   1:  PR[GP1:91,2] = PR[GP1:90,2] + -18.164;
   1:L PR[91] 10mm/sec CNT100;
   1:  PR[GP1:91,1] = PR[GP1:90,1] + -12.359;
   1:  PR[GP1:91,2] = PR[GP1:90,2] + -17.916;
   1:L PR[91] 10mm/sec CNT100;
   1:  PR[GP1:91,1] = PR[GP1:90,1] + -10.331;
   1:  PR[GP1:91,2] = PR[GP1:90,2] + -17.601;
   1:L PR[91] 10mm/sec CNT100;
   1:  PR[GP1:91,1] = PR[GP1:90,1] + -9.404;
   1:  PR[GP1:91,2] = PR[GP1:90,2] + -17.336;
   1:L PR[91] 10mm/sec CNT100;
   1:  PR[GP1:91,1] = PR[GP1:90,1] + -7.263;
   1:  PR[GP1:91,2] = PR[GP1:90,2] + -16.549;
   1:L PR[91] 10mm/sec CNT100;
   1:  PR[GP1:91,1] = PR[GP1:90,1] + -5.060;
   1:  PR[GP1:91,2] = PR[GP1:90,2] + -15.429;
   1:L PR[91] 10mm/sec CNT100;
   1:  PR[GP1:91,1] = PR[GP1:90,1] + -4.584;
   1:  PR[GP1:91,2] = PR[GP1:90,2] + -15.127;
   1:L PR[91] 10mm/sec CNT100;
   1:  PR[GP1:91,1] = PR[GP1:90,1] + -3.585;
   1:  PR[GP1:91,2] = PR[GP1:90,2] + -14.315;
   1:L PR[91] 10mm/sec CNT100;
   1:  PR[GP1:91,1] = PR[GP1:90,1] + -2.076;
   1:  PR[GP1:91,2] = PR[GP1:90,2] + -13.237;
   1:L PR[91] 10mm/sec CNT100;
   1:  PR[GP1:91,1] = PR[GP1:90,1] + -1.387;
   1:  PR[GP1:91,2] = PR[GP1:90,2] + -12.844;
   1:L PR[91] 10mm/sec CNT100;
   1:  PR[GP1:91,1] = PR[GP1:90,1] + -1.119;
   1:  PR[GP1:91,2] = PR[GP1:90,2] + -12.728;
   1:L PR[91] 10mm/sec CNT100;
   1:  PR[GP1:91,1] = PR[GP1:90,1] + -0.823;
   1:  PR[GP1:91,2] = PR[GP1:90,2] + -12.708;
   1:L PR[91] 10mm/sec CNT100;
   1:  PR[GP1:91,1] = PR[GP1:90,1] + -0.008;
   1:  PR[GP1:91,2] = PR[GP1:90,2] + -12.753;
   1:L PR[91] 10mm/sec CNT100;
   1:  PR[GP1:91,1] = PR[GP1:90,1] + 0.309;
   1:  PR[GP1:91,2] = PR[GP1:90,2] + -12.841;
   1:L PR[91] 10mm/sec CNT100;
   1:  PR[GP1:91,1] = PR[GP1:90,1] + 0.588;
   1:  PR[GP1:91,2] = PR[GP1:90,2] + -13.019;
   1:L PR[91] 10mm/sec CNT100;
   1:  PR[GP1:91,1] = PR[GP1:90,1] + 0.819;
   1:  PR[GP1:91,2] = PR[GP1:90,2] + -13.215;
   1:L PR[91] 10mm/sec CNT100;
   1:  PR[GP1:91,1] = PR[GP1:90,1] + 1.159;
   1:  PR[GP1:91,2] = PR[GP1:90,2] + -13.460;
   1:L PR[91] 10mm/sec CNT100;
   1:  PR[GP1:91,1] = PR[GP1:90,1] + 1.845;
   1:  PR[GP1:91,2] = PR[GP1:90,2] + -14.074;
   1:L PR[91] 10mm/sec CNT100;
   1:  PR[GP1:91,1] = PR[GP1:90,1] + 3.504;
   1:  PR[GP1:91,2] = PR[GP1:90,2] + -15.397;
   1:L PR[91] 10mm/sec CNT100;
   1:  PR[GP1:91,1] = PR[GP1:90,1] + 4.173;
   1:  PR[GP1:91,2] = PR[GP1:90,2] + -15.810;
   1:L PR[91] 10mm/sec CNT100;
   1:  PR[GP1:91,1] = PR[GP1:90,1] + 5.723;
   1:  PR[GP1:91,2] = PR[GP1:90,2] + -16.693;
   1:L PR[91] 10mm/sec CNT100;
   1:  PR[GP1:91,1] = PR[GP1:90,1] + 6.877;
   1:  PR[GP1:91,2] = PR[GP1:90,2] + -17.178;
   1:L PR[91] 10mm/sec CNT100;
   1:  PR[GP1:91,1] = PR[GP1:90,1] + 8.132;
   1:  PR[GP1:91,2] = PR[GP1:90,2] + -17.659;
   1:L PR[91] 10mm/sec CNT100;
   1:  PR[GP1:91,1] = PR[GP1:90,1] + 9.969;
   1:  PR[GP1:91,2] = PR[GP1:90,2] + -18.120;
   1:L PR[91] 10mm/sec CNT100;
   1:  PR[GP1:91,1] = PR[GP1:90,1] + 10.684;
   1:  PR[GP1:91,2] = PR[GP1:90,2] + -18.278;
   1:L PR[91] 10mm/sec CNT100;
   1:  PR[GP1:91,1] = PR[GP1:90,1] + 13.342;
   1:  PR[GP1:91,2] = PR[GP1:90,2] + -18.537;
   1:L PR[91] 10mm/sec CNT100;
   1:  PR[GP1:91,1] = PR[GP1:90,1] + 16.066;
   1:  PR[GP1:91,2] = PR[GP1:90,2] + -18.455;
   1:L PR[91] 10mm/sec CNT100;
   1:  PR[GP1:91,1] = PR[GP1:90,1] + 17.172;
   1:  PR[GP1:91,2] = PR[GP1:90,2] + -18.288;
   1:L PR[91] 10mm/sec CNT100;
   1:  PR[GP1:91,1] = PR[GP1:90,1] + 18.772;
   1:  PR[GP1:91,2] = PR[GP1:90,2] + -18.012;
   1:L PR[91] 10mm/sec CNT100;
   1:  PR[GP1:91,1] = PR[GP1:90,1] + 21.428;
   1:  PR[GP1:91,2] = PR[GP1:90,2] + -17.205;
   1:L PR[91] 10mm/sec CNT100;
   1:  PR[GP1:91,1] = PR[GP1:90,1] + 22.270;
   1:  PR[GP1:91,2] = PR[GP1:90,2] + -16.815;
   1:L PR[91] 10mm/sec CNT100;
   1:  PR[GP1:91,1] = PR[GP1:90,1] + 23.997;
   1:  PR[GP1:91,2] = PR[GP1:90,2] + -16.051;
   1:L PR[91] 10mm/sec CNT100;
   1:  PR[GP1:91,1] = PR[GP1:90,1] + 26.389;
   1:  PR[GP1:91,2] = PR[GP1:90,2] + -14.564;
   1:L PR[91] 10mm/sec CNT100;
   1:  PR[GP1:91,1] = PR[GP1:90,1] + 28.540;
   1:  PR[GP1:91,2] = PR[GP1:90,2] + -12.759;
   1:L PR[91] 10mm/sec CNT100;
   1:  PR[GP1:91,1] = PR[GP1:90,1] + 30.389;
   1:  PR[GP1:91,2] = PR[GP1:90,2] + -10.671;
   1:L PR[91] 10mm/sec CNT100;
   1:  PR[GP1:91,1] = PR[GP1:90,1] + 31.864;
   1:  PR[GP1:91,2] = PR[GP1:90,2] + -8.345;
   1:L PR[91] 10mm/sec CNT100;
   1:  PR[GP1:91,1] = PR[GP1:90,1] + 32.941;
   1:  PR[GP1:91,2] = PR[GP1:90,2] + -5.850;
   1:L PR[91] 10mm/sec CNT100;
   1:  PR[GP1:91,1] = PR[GP1:90,1] + 33.595;
   1:  PR[GP1:91,2] = PR[GP1:90,2] + -3.244;
   1:L PR[91] 10mm/sec CNT100;
   1:  PR[GP1:91,1] = PR[GP1:90,1] + 33.828;
   1:  PR[GP1:91,2] = PR[GP1:90,2] + -0.590;
   1:L PR[91] 10mm/sec CNT100;
   1:  PR[GP1:91,1] = PR[GP1:90,1] + 33.694;
   1:  PR[GP1:91,2] = PR[GP1:90,2] + 0.668;
   1:L PR[91] 10mm/sec CNT100;
   1:  PR[GP1:91,1] = PR[GP1:90,1] + 33.448;
   1:  PR[GP1:91,2] = PR[GP1:90,2] + 2.737;
   1:L PR[91] 10mm/sec CNT100;
   1:  PR[GP1:91,1] = PR[GP1:90,1] + 32.398;
   1:  PR[GP1:91,2] = PR[GP1:90,2] + 5.926;
   1:L PR[91] 10mm/sec CNT100;
   1:  PR[GP1:91,1] = PR[GP1:90,1] + 30.698;
   1:  PR[GP1:91,2] = PR[GP1:90,2] + 8.848;
   1:L PR[91] 10mm/sec CNT100;
   1:  PR[GP1:91,1] = PR[GP1:90,1] + 28.399;
   1:  PR[GP1:91,2] = PR[GP1:90,2] + 11.386;
   1:L PR[91] 10mm/sec CNT100;
   1:  PR[GP1:91,1] = PR[GP1:90,1] + 25.561;
   1:  PR[GP1:91,2] = PR[GP1:90,2] + 13.437;
   1:L PR[91] 10mm/sec CNT100;
   1:  PR[GP1:91,1] = PR[GP1:90,1] + 22.318;
   1:  PR[GP1:91,2] = PR[GP1:90,2] + 14.932;
   1:L PR[91] 10mm/sec CNT100;
   1:  PR[GP1:91,1] = PR[GP1:90,1] + 20.352;
   1:  PR[GP1:91,2] = PR[GP1:90,2] + 15.425;
   1:L PR[91] 10mm/sec CNT100;
   1:  PR[GP1:91,1] = PR[GP1:90,1] + 18.805;
   1:  PR[GP1:91,2] = PR[GP1:90,2] + 15.794;
   1:L PR[91] 10mm/sec CNT100;
   1:  PR[GP1:91,1] = PR[GP1:90,1] + 15.138;
   1:  PR[GP1:91,2] = PR[GP1:90,2] + 15.989;
   1:L PR[91] 10mm/sec CNT100;
   1:  PR[GP1:91,1] = PR[GP1:90,1] + 11.469;
   1:  PR[GP1:91,2] = PR[GP1:90,2] + 15.530;
   1:L PR[91] 10mm/sec CNT100;
   1:  PR[GP1:91,1] = PR[GP1:90,1] + 7.988;
   1:  PR[GP1:91,2] = PR[GP1:90,2] + 14.405;
   1:L PR[91] 10mm/sec CNT100;
   1:  PR[GP1:91,1] = PR[GP1:90,1] + 4.755;
   1:  PR[GP1:91,2] = PR[GP1:90,2] + 12.699;
   1:L PR[91] 10mm/sec CNT100;
   1:  PR[GP1:91,1] = PR[GP1:90,1] + 1.964;
   1:  PR[GP1:91,2] = PR[GP1:90,2] + 10.434;
   1:L PR[91] 10mm/sec CNT100;
   1:  PR[GP1:91,1] = PR[GP1:90,1] + 1.006;
   1:  PR[GP1:91,2] = PR[GP1:90,2] + 9.382;
   1:L PR[91] 10mm/sec CNT100;
   1:  PR[GP1:91,1] = PR[GP1:90,1] + -0.059;
   1:  PR[GP1:91,2] = PR[GP1:90,2] + 8.752;
   1:L PR[91] 10mm/sec CNT100;
   1:  PR[GP1:91,1] = PR[GP1:90,1] + -1.331;
   1:  PR[GP1:91,2] = PR[GP1:90,2] + 8.647;
   1:L PR[91] 10mm/sec CNT100;
   1:  PR[GP1:91,1] = PR[GP1:90,1] + -2.491;
   1:  PR[GP1:91,2] = PR[GP1:90,2] + 9.147;
   1:L PR[91] 10mm/sec CNT100;
   1:  PR[GP1:91,1] = PR[GP1:90,1] + -2.719;
   1:  PR[GP1:91,2] = PR[GP1:90,2] + 9.381;
   1:L PR[91] 10mm/sec CNT100;
   1:  PR[GP1:91,1] = PR[GP1:90,1] + -4.261;
   1:  PR[GP1:91,2] = PR[GP1:90,2] + 10.720;
   1:L PR[91] 10mm/sec CNT100;
   1:  PR[GP1:91,1] = PR[GP1:90,1] + -4.987;
   1:  PR[GP1:91,2] = PR[GP1:90,2] + 11.416;
   1:L PR[91] 10mm/sec CNT100;
   1:  PR[GP1:91,1] = PR[GP1:90,1] + -5.273;
   1:  PR[GP1:91,2] = PR[GP1:90,2] + 11.663;
   1:L PR[91] 10mm/sec CNT100;
   1:  PR[GP1:91,1] = PR[GP1:90,1] + -7.389;
   1:  PR[GP1:91,2] = PR[GP1:90,2] + 13.010;
   1:L PR[91] 10mm/sec CNT100;
   1:  PR[GP1:91,1] = PR[GP1:90,1] + -8.747;
   1:  PR[GP1:91,2] = PR[GP1:90,2] + 13.793;
   1:L PR[91] 10mm/sec CNT100;
   1:  PR[GP1:91,1] = PR[GP1:90,1] + -10.045;
   1:  PR[GP1:91,2] = PR[GP1:90,2] + 14.305;
   1:L PR[91] 10mm/sec CNT100;
   1:  PR[GP1:91,1] = PR[GP1:90,1] + -12.511;
   1:  PR[GP1:91,2] = PR[GP1:90,2] + 15.171;
   1:L PR[91] 10mm/sec CNT100;
   1:  PR[GP1:91,1] = PR[GP1:90,1] + -12.926;
   1:  PR[GP1:91,2] = PR[GP1:90,2] + 15.249;
   1:L PR[91] 10mm/sec CNT100;
   1:  PR[GP1:91,1] = PR[GP1:90,1] + -16.261;
   1:  PR[GP1:91,2] = PR[GP1:90,2] + 15.760;
   1:L PR[91] 10mm/sec CNT100;
   1:  PR[GP1:91,1] = PR[GP1:90,1] + -19.861;
   1:  PR[GP1:91,2] = PR[GP1:90,2] + 15.600;
   1:L PR[91] 10mm/sec CNT100;
   1:  PR[GP1:91,1] = PR[GP1:90,1] + -23.311;
   1:  PR[GP1:91,2] = PR[GP1:90,2] + 14.747;
   1:L PR[91] 10mm/sec CNT100;
   1:  PR[GP1:91,1] = PR[GP1:90,1] + -26.480;
   1:  PR[GP1:91,2] = PR[GP1:90,2] + 13.247;
   1:L PR[91] 10mm/sec CNT100;
   1:  PR[GP1:91,1] = PR[GP1:90,1] + -27.535;
   1:  PR[GP1:91,2] = PR[GP1:90,2] + 12.459;
   1:L PR[91] 10mm/sec CNT100;
   1:  PR[GP1:91,1] = PR[GP1:90,1] + -29.240;
   1:  PR[GP1:91,2] = PR[GP1:90,2] + 11.168;
   1:L PR[91] 10mm/sec CNT100;
   1:  PR[GP1:91,1] = PR[GP1:90,1] + -31.489;
   1:  PR[GP1:91,2] = PR[GP1:90,2] + 8.592;
   1:L PR[91] 10mm/sec CNT100;
   1:  PR[GP1:91,1] = PR[GP1:90,1] + -33.148;
   1:  PR[GP1:91,2] = PR[GP1:90,2] + 5.626;
   1:L PR[91] 10mm/sec CNT100;
   1:  PR[GP1:91,1] = PR[GP1:90,1] + -34.167;
   1:  PR[GP1:91,2] = PR[GP1:90,2] + 2.399;
   1:L PR[91] 10mm/sec CNT100;
   1:  PR[GP1:91,1] = PR[GP1:90,1] + -34.462;
   1:  PR[GP1:91,2] = PR[GP1:90,2] + -0.988;
   1:L PR[91] 10mm/sec CNT100;
   1:  PR[GP1:91,1] = PR[GP1:90,1] + -34.182;
   1:  PR[GP1:91,2] = PR[GP1:90,2] + -3.284;
   1:L PR[91] 10mm/sec CNT100;
   1:  PR[GP1:91,1] = PR[GP1:90,1] + -34.029;
   1:  PR[GP1:91,2] = PR[GP1:90,2] + -4.407;
   1:L PR[91] 10mm/sec CNT100;
   1:  PR[GP1:91,1] = PR[GP1:90,1] + -32.928;
   1:  PR[GP1:91,2] = PR[GP1:90,2] + -7.698;
   1:L PR[91] 10mm/sec CNT100;
   1:  PR[GP1:91,1] = PR[GP1:90,1] + -31.996;
   1:  PR[GP1:91,2] = PR[GP1:90,2] + -9.300;
   1:L PR[91] 10mm/sec CNT100;
   1:  PR[GP1:91,1] = PR[GP1:90,1] + -31.134;
   1:  PR[GP1:91,2] = PR[GP1:90,2] + -10.741;
   1:L PR[91] 10mm/sec CNT100;
   1:  PR[GP1:91,1] = PR[GP1:90,1] + -30.170;
   1:  PR[GP1:91,2] = PR[GP1:90,2] + -11.828;
   1:L PR[91] 10mm/sec CNT100;
   1:  PR[GP1:91,1] = PR[GP1:90,1] + -28.716;
   1:  PR[GP1:91,2] = PR[GP1:90,2] + -13.413;
   1:L PR[91] 10mm/sec CNT100;
   1:  PR[GP1:91,1] = PR[GP1:90,1] + -27.974;
   1:  PR[GP1:91,2] = PR[GP1:90,2] + -13.976;
   1:L PR[91] 10mm/sec CNT100;
   1:  PR[GP1:91,1] = PR[GP1:90,1] + -25.772;
   1:  PR[GP1:91,2] = PR[GP1:90,2] + -15.582;
   1:L PR[91] 10mm/sec CNT100;
   1:  PR[GP1:91,1] = PR[GP1:90,1] + -22.686;
   1:  PR[GP1:91,2] = PR[GP1:90,2] + -16.956;
   1:  PR[GP1:91,3] = PR[GP1:90,3] + 22.000;
   1:L PR[91] 10mm/sec CNT100;
   1:  PR[GP1:91,1] = PR[GP1:90,1] + -21.626;
   1:  PR[GP1:91,2] = PR[GP1:90,2] + -17.393;
   1:L PR[91] 10mm/sec CNT100;
   1:  PR[GP1:91,1] = PR[GP1:90,1] + -19.736;
   1:  PR[GP1:91,2] = PR[GP1:90,2] + -17.865;
   1:L PR[91] 10mm/sec CNT100;
   1:  PR[GP1:91,1] = PR[GP1:90,1] + -17.575;
   1:  PR[GP1:91,2] = PR[GP1:90,2] + -18.300;
   1:L PR[91] 10mm/sec CNT100;
   1:  PR[GP1:91,1] = PR[GP1:90,1] + -16.748;
   1:  PR[GP1:91,2] = PR[GP1:90,2] + -18.347;
   1:L PR[91] 10mm/sec CNT100;
   1:  PR[GP1:91,1] = PR[GP1:90,1] + -14.549;
   1:  PR[GP1:91,2] = PR[GP1:90,2] + -18.356;
   1:L PR[91] 10mm/sec CNT100;
   1:  PR[GP1:91,1] = PR[GP1:90,1] + -13.511;
   1:  PR[GP1:91,2] = PR[GP1:90,2] + -18.391;
   1:L PR[91] 10mm/sec CNT100;
   1:  PR[GP1:91,1] = PR[GP1:90,1] + -13.019;
   1:  PR[GP1:91,2] = PR[GP1:90,2] + -18.345;
   1:L PR[91] 10mm/sec CNT100;
   1:  PR[GP1:91,1] = PR[GP1:90,1] + -10.139;
   1:  PR[GP1:91,2] = PR[GP1:90,2] + -17.896;
   1:L PR[91] 10mm/sec CNT100;
   1:  PR[GP1:91,1] = PR[GP1:90,1] + -7.967;
   1:  PR[GP1:91,2] = PR[GP1:90,2] + -17.277;
   1:L PR[91] 10mm/sec CNT100;
   1:  PR[GP1:91,1] = PR[GP1:90,1] + -7.115;
   1:  PR[GP1:91,2] = PR[GP1:90,2] + -16.963;
   1:L PR[91] 10mm/sec CNT100;
   1:  PR[GP1:91,1] = PR[GP1:90,1] + -5.548;
   1:  PR[GP1:91,2] = PR[GP1:90,2] + -16.167;
   1:L PR[91] 10mm/sec CNT100;
   1:  PR[GP1:91,1] = PR[GP1:90,1] + -4.227;
   1:  PR[GP1:91,2] = PR[GP1:90,2] + -15.588;
   1:L PR[91] 10mm/sec CNT100;
   1:  PR[GP1:91,1] = PR[GP1:90,1] + -3.745;
   1:  PR[GP1:91,2] = PR[GP1:90,2] + -15.309;
   1:L PR[91] 10mm/sec CNT100;
   1:  PR[GP1:91,1] = PR[GP1:90,1] + -1.814;
   1:  PR[GP1:91,2] = PR[GP1:90,2] + -13.929;
   1:L PR[91] 10mm/sec CNT100;
   1:  PR[GP1:91,1] = PR[GP1:90,1] + -1.357;
   1:  PR[GP1:91,2] = PR[GP1:90,2] + -13.668;
   1:L PR[91] 10mm/sec CNT100;
   1:  PR[GP1:91,1] = PR[GP1:90,1] + -0.946;
   1:  PR[GP1:91,2] = PR[GP1:90,2] + -13.490;
   1:L PR[91] 10mm/sec CNT100;
   1:  PR[GP1:91,1] = PR[GP1:90,1] + -0.492;
   1:  PR[GP1:91,2] = PR[GP1:90,2] + -13.460;
   1:L PR[91] 10mm/sec CNT100;
   1:  PR[GP1:91,1] = PR[GP1:90,1] + 0.060;
   1:  PR[GP1:91,2] = PR[GP1:90,2] + -13.490;
   1:L PR[91] 10mm/sec CNT100;
   1:  PR[GP1:91,1] = PR[GP1:90,1] + 0.533;
   1:  PR[GP1:91,2] = PR[GP1:90,2] + -13.622;
   1:L PR[91] 10mm/sec CNT100;
   1:  PR[GP1:91,1] = PR[GP1:90,1] + 0.971;
   1:  PR[GP1:91,2] = PR[GP1:90,2] + -13.902;
   1:L PR[91] 10mm/sec CNT100;
   1:  PR[GP1:91,1] = PR[GP1:90,1] + 1.295;
   1:  PR[GP1:91,2] = PR[GP1:90,2] + -14.177;
   1:L PR[91] 10mm/sec CNT100;
   1:  PR[GP1:91,1] = PR[GP1:90,1] + 3.201;
   1:  PR[GP1:91,2] = PR[GP1:90,2] + -15.686;
   1:L PR[91] 10mm/sec CNT100;
   1:  PR[GP1:91,1] = PR[GP1:90,1] + 5.442;
   1:  PR[GP1:91,2] = PR[GP1:90,2] + -16.966;
   1:L PR[91] 10mm/sec CNT100;
   1:  PR[GP1:91,1] = PR[GP1:90,1] + 5.833;
   1:  PR[GP1:91,2] = PR[GP1:90,2] + -17.130;
   1:L PR[91] 10mm/sec CNT100;
   1:  PR[GP1:91,1] = PR[GP1:90,1] + 7.860;
   1:  PR[GP1:91,2] = PR[GP1:90,2] + -17.907;
   1:L PR[91] 10mm/sec CNT100;
   1:  PR[GP1:91,1] = PR[GP1:90,1] + 8.824;
   1:  PR[GP1:91,2] = PR[GP1:90,2] + -18.149;
   1:L PR[91] 10mm/sec CNT100;
   1:  PR[GP1:91,1] = PR[GP1:90,1] + 10.416;
   1:  PR[GP1:91,2] = PR[GP1:90,2] + -18.502;
   1:L PR[91] 10mm/sec CNT100;
   1:  PR[GP1:91,1] = PR[GP1:90,1] + 12.160;
   1:  PR[GP1:91,2] = PR[GP1:90,2] + -18.671;
   1:L PR[91] 10mm/sec CNT100;
   1:  PR[GP1:91,1] = PR[GP1:90,1] + 13.059;
   1:  PR[GP1:91,2] = PR[GP1:90,2] + -18.737;
   1:L PR[91] 10mm/sec CNT100;
   1:  PR[GP1:91,1] = PR[GP1:90,1] + 15.753;
   1:  PR[GP1:91,2] = PR[GP1:90,2] + -18.605;
   1:L PR[91] 10mm/sec CNT100;
   1:  PR[GP1:91,1] = PR[GP1:90,1] + 18.461;
   1:  PR[GP1:91,2] = PR[GP1:90,2] + -18.137;
   1:L PR[91] 10mm/sec CNT100;
   1:  PR[GP1:91,1] = PR[GP1:90,1] + 19.568;
   1:  PR[GP1:91,2] = PR[GP1:90,2] + -17.804;
   1:L PR[91] 10mm/sec CNT100;
   1:  PR[GP1:91,1] = PR[GP1:90,1] + 21.096;
   1:  PR[GP1:91,2] = PR[GP1:90,2] + -17.314;
   1:L PR[91] 10mm/sec CNT100;
   1:  PR[GP1:91,1] = PR[GP1:90,1] + 23.318;
   1:  PR[GP1:91,2] = PR[GP1:90,2] + -16.284;
   1:L PR[91] 10mm/sec CNT100;
   1:  PR[GP1:91,1] = PR[GP1:90,1] + 23.620;
   1:  PR[GP1:91,2] = PR[GP1:90,2] + -16.138;
   1:L PR[91] 10mm/sec CNT100;
   1:  PR[GP1:91,1] = PR[GP1:90,1] + 25.995;
   1:  PR[GP1:91,2] = PR[GP1:90,2] + -14.632;
   1:L PR[91] 10mm/sec CNT100;
   1:  PR[GP1:91,1] = PR[GP1:90,1] + 28.131;
   1:  PR[GP1:91,2] = PR[GP1:90,2] + -12.821;
   1:L PR[91] 10mm/sec CNT100;
   1:  PR[GP1:91,1] = PR[GP1:90,1] + 29.968;
   1:  PR[GP1:91,2] = PR[GP1:90,2] + -10.732;
   1:L PR[91] 10mm/sec CNT100;
   1:  PR[GP1:91,1] = PR[GP1:90,1] + 31.456;
   1:  PR[GP1:91,2] = PR[GP1:90,2] + -8.409;
   1:L PR[91] 10mm/sec CNT100;
   1:  PR[GP1:91,1] = PR[GP1:90,1] + 31.914;
   1:  PR[GP1:91,2] = PR[GP1:90,2] + -7.365;
   1:L PR[91] 10mm/sec CNT100;
   1:  PR[GP1:91,1] = PR[GP1:90,1] + 32.539;
   1:  PR[GP1:91,2] = PR[GP1:90,2] + -5.912;
   1:L PR[91] 10mm/sec CNT100;
   1:  PR[GP1:91,1] = PR[GP1:90,1] + 33.191;
   1:  PR[GP1:91,2] = PR[GP1:90,2] + -3.302;
   1:L PR[91] 10mm/sec CNT100;
   1:  PR[GP1:91,1] = PR[GP1:90,1] + 33.407;
   1:  PR[GP1:91,2] = PR[GP1:90,2] + -0.645;
   1:L PR[91] 10mm/sec CNT100;
   1:  PR[GP1:91,1] = PR[GP1:90,1] + 33.051;
   1:  PR[GP1:91,2] = PR[GP1:90,2] + 2.698;
   1:L PR[91] 10mm/sec CNT100;
   1:  PR[GP1:91,1] = PR[GP1:90,1] + 31.990;
   1:  PR[GP1:91,2] = PR[GP1:90,2] + 5.880;
   1:L PR[91] 10mm/sec CNT100;
   1:  PR[GP1:91,1] = PR[GP1:90,1] + 30.259;
   1:  PR[GP1:91,2] = PR[GP1:90,2] + 8.792;
   1:L PR[91] 10mm/sec CNT100;
   1:  PR[GP1:91,1] = PR[GP1:90,1] + 27.925;
   1:  PR[GP1:91,2] = PR[GP1:90,2] + 11.324;
   1:L PR[91] 10mm/sec CNT100;
   1:  PR[GP1:91,1] = PR[GP1:90,1] + 25.080;
   1:  PR[GP1:91,2] = PR[GP1:90,2] + 13.376;
   1:L PR[91] 10mm/sec CNT100;
   1:  PR[GP1:91,1] = PR[GP1:90,1] + 21.838;
   1:  PR[GP1:91,2] = PR[GP1:90,2] + 14.866;
   1:L PR[91] 10mm/sec CNT100;
   1:  PR[GP1:91,1] = PR[GP1:90,1] + 18.310;
   1:  PR[GP1:91,2] = PR[GP1:90,2] + 15.707;
   1:L PR[91] 10mm/sec CNT100;
   1:  PR[GP1:91,1] = PR[GP1:90,1] + 16.817;
   1:  PR[GP1:91,2] = PR[GP1:90,2] + 15.790;
   1:L PR[91] 10mm/sec CNT100;
   1:  PR[GP1:91,1] = PR[GP1:90,1] + 14.649;
   1:  PR[GP1:91,2] = PR[GP1:90,2] + 15.896;
   1:L PR[91] 10mm/sec CNT100;
   1:  PR[GP1:91,1] = PR[GP1:90,1] + 12.630;
   1:  PR[GP1:91,2] = PR[GP1:90,2] + 15.644;
   1:L PR[91] 10mm/sec CNT100;
   1:  PR[GP1:91,1] = PR[GP1:90,1] + 11.012;
   1:  PR[GP1:91,2] = PR[GP1:90,2] + 15.420;
   1:L PR[91] 10mm/sec CNT100;
   1:  PR[GP1:91,1] = PR[GP1:90,1] + 7.526;
   1:  PR[GP1:91,2] = PR[GP1:90,2] + 14.295;
   1:L PR[91] 10mm/sec CNT100;
   1:  PR[GP1:91,1] = PR[GP1:90,1] + 5.481;
   1:  PR[GP1:91,2] = PR[GP1:90,2] + 13.217;
   1:L PR[91] 10mm/sec CNT100;
   1:  PR[GP1:91,1] = PR[GP1:90,1] + 4.329;
   1:  PR[GP1:91,2] = PR[GP1:90,2] + 12.582;
   1:L PR[91] 10mm/sec CNT100;
   1:  PR[GP1:91,1] = PR[GP1:90,1] + 1.517;
   1:  PR[GP1:91,2] = PR[GP1:90,2] + 10.318;
   1:L PR[91] 10mm/sec CNT100;
   1:  PR[GP1:91,1] = PR[GP1:90,1] + 1.015;
   1:  PR[GP1:91,2] = PR[GP1:90,2] + 9.766;
   1:L PR[91] 10mm/sec CNT100;
   1:  PR[GP1:91,1] = PR[GP1:90,1] + 0.540;
   1:  PR[GP1:91,2] = PR[GP1:90,2] + 9.487;
   1:L PR[91] 10mm/sec CNT100;
   1:  PR[GP1:91,1] = PR[GP1:90,1] + -0.010;
   1:  PR[GP1:91,2] = PR[GP1:90,2] + 9.110;
   1:L PR[91] 10mm/sec CNT100;
   1:  PR[GP1:91,1] = PR[GP1:90,1] + -0.917;
   1:  PR[GP1:91,2] = PR[GP1:90,2] + 9.035;
   1:L PR[91] 10mm/sec CNT100;
   1:  PR[GP1:91,1] = PR[GP1:90,1] + -1.387;
   1:  PR[GP1:91,2] = PR[GP1:90,2] + 9.039;
   1:L PR[91] 10mm/sec CNT100;
   1:  PR[GP1:91,1] = PR[GP1:90,1] + -2.129;
   1:  PR[GP1:91,2] = PR[GP1:90,2] + 9.457;
   1:L PR[91] 10mm/sec CNT100;
   1:  PR[GP1:91,1] = PR[GP1:90,1] + -2.468;
   1:  PR[GP1:91,2] = PR[GP1:90,2] + 9.604;
   1:L PR[91] 10mm/sec CNT100;
   1:  PR[GP1:91,1] = PR[GP1:90,1] + -4.460;
   1:  PR[GP1:91,2] = PR[GP1:90,2] + 11.333;
   1:L PR[91] 10mm/sec CNT100;
   1:  PR[GP1:91,1] = PR[GP1:90,1] + -4.856;
   1:  PR[GP1:91,2] = PR[GP1:90,2] + 11.606;
   1:L PR[91] 10mm/sec CNT100;
   1:  PR[GP1:91,1] = PR[GP1:90,1] + -5.842;
   1:  PR[GP1:91,2] = PR[GP1:90,2] + 12.188;
   1:L PR[91] 10mm/sec CNT100;
   1:  PR[GP1:91,1] = PR[GP1:90,1] + -7.468;
   1:  PR[GP1:91,2] = PR[GP1:90,2] + 13.223;
   1:L PR[91] 10mm/sec CNT100;
   1:  PR[GP1:91,1] = PR[GP1:90,1] + -8.098;
   1:  PR[GP1:91,2] = PR[GP1:90,2] + 13.586;
   1:L PR[91] 10mm/sec CNT100;
   1:  PR[GP1:91,1] = PR[GP1:90,1] + -10.151;
   1:  PR[GP1:91,2] = PR[GP1:90,2] + 14.395;
   1:L PR[91] 10mm/sec CNT100;
   1:  PR[GP1:91,1] = PR[GP1:90,1] + -11.888;
   1:  PR[GP1:91,2] = PR[GP1:90,2] + 15.005;
   1:L PR[91] 10mm/sec CNT100;
   1:  PR[GP1:91,1] = PR[GP1:90,1] + -13.037;
   1:  PR[GP1:91,2] = PR[GP1:90,2] + 15.222;
   1:L PR[91] 10mm/sec CNT100;
   1:  PR[GP1:91,1] = PR[GP1:90,1] + -15.778;
   1:  PR[GP1:91,2] = PR[GP1:90,2] + 15.645;
   1:L PR[91] 10mm/sec CNT100;
   1:  PR[GP1:91,1] = PR[GP1:90,1] + -17.595;
   1:  PR[GP1:91,2] = PR[GP1:90,2] + 15.595;
   1:L PR[91] 10mm/sec CNT100;
   1:  PR[GP1:91,1] = PR[GP1:90,1] + -19.495;
   1:  PR[GP1:91,2] = PR[GP1:90,2] + 15.513;
   1:L PR[91] 10mm/sec CNT100;
   1:  PR[GP1:91,1] = PR[GP1:90,1] + -22.956;
   1:  PR[GP1:91,2] = PR[GP1:90,2] + 14.663;
   1:L PR[91] 10mm/sec CNT100;
   1:  PR[GP1:91,1] = PR[GP1:90,1] + -26.134;
   1:  PR[GP1:91,2] = PR[GP1:90,2] + 13.163;
   1:L PR[91] 10mm/sec CNT100;
   1:  PR[GP1:91,1] = PR[GP1:90,1] + -27.631;
   1:  PR[GP1:91,2] = PR[GP1:90,2] + 12.045;
   1:L PR[91] 10mm/sec CNT100;
   1:  PR[GP1:91,1] = PR[GP1:90,1] + -28.903;
   1:  PR[GP1:91,2] = PR[GP1:90,2] + 11.082;
   1:L PR[91] 10mm/sec CNT100;
   1:  PR[GP1:91,1] = PR[GP1:90,1] + -31.158;
   1:  PR[GP1:91,2] = PR[GP1:90,2] + 8.502;
   1:L PR[91] 10mm/sec CNT100;
   1:  PR[GP1:91,1] = PR[GP1:90,1] + -32.821;
   1:  PR[GP1:91,2] = PR[GP1:90,2] + 5.530;
   1:L PR[91] 10mm/sec CNT100;
   1:  PR[GP1:91,1] = PR[GP1:90,1] + -33.844;
   1:  PR[GP1:91,2] = PR[GP1:90,2] + 2.298;
   1:L PR[91] 10mm/sec CNT100;
   1:  PR[GP1:91,1] = PR[GP1:90,1] + -34.140;
   1:  PR[GP1:91,2] = PR[GP1:90,2] + -1.095;
   1:L PR[91] 10mm/sec CNT100;
   1:  PR[GP1:91,1] = PR[GP1:90,1] + -33.930;
   1:  PR[GP1:91,2] = PR[GP1:90,2] + -2.827;
   1:L PR[91] 10mm/sec CNT100;
   1:  PR[GP1:91,1] = PR[GP1:90,1] + -33.698;
   1:  PR[GP1:91,2] = PR[GP1:90,2] + -4.526;
   1:L PR[91] 10mm/sec CNT100;
   1:  PR[GP1:91,1] = PR[GP1:90,1] + -32.591;
   1:  PR[GP1:91,2] = PR[GP1:90,2] + -7.826;
   1:L PR[91] 10mm/sec CNT100;
   1:  PR[GP1:91,1] = PR[GP1:90,1] + -31.940;
   1:  PR[GP1:91,2] = PR[GP1:90,2] + -8.946;
   1:L PR[91] 10mm/sec CNT100;
   1:  PR[GP1:91,1] = PR[GP1:90,1] + -30.784;
   1:  PR[GP1:91,2] = PR[GP1:90,2] + -10.878;
   1:L PR[91] 10mm/sec CNT100;
   1:  PR[GP1:91,1] = PR[GP1:90,1] + -30.206;
   1:  PR[GP1:91,2] = PR[GP1:90,2] + -11.529;
   1:L PR[91] 10mm/sec CNT100;
   1:  PR[GP1:91,1] = PR[GP1:90,1] + -28.351;
   1:  PR[GP1:91,2] = PR[GP1:90,2] + -13.551;
   1:L PR[91] 10mm/sec CNT100;
   1:  PR[GP1:91,1] = PR[GP1:90,1] + -26.649;
   1:  PR[GP1:91,2] = PR[GP1:90,2] + -14.802;
   1:L PR[91] 10mm/sec CNT100;
   1:  PR[GP1:91,1] = PR[GP1:90,1] + -25.295;
   1:  PR[GP1:91,2] = PR[GP1:90,2] + -15.755;
   1:L PR[91] 10mm/sec CNT100;
   1:  PR[GP1:91,1] = PR[GP1:90,1] + -24.714;
   1:  PR[GP1:91,2] = PR[GP1:90,2] + -15.966;
   1:  PR[GP1:91,3] = PR[GP1:90,3] + 23.100;
   1:L PR[91] 10mm/sec CNT100;
   1:  PR[GP1:91,1] = PR[GP1:90,1] + -22.739;
   1:  PR[GP1:91,2] = PR[GP1:90,2] + -16.875;
   1:L PR[91] 10mm/sec CNT100;
   1:  PR[GP1:91,1] = PR[GP1:90,1] + -20.987;
   1:  PR[GP1:91,2] = PR[GP1:90,2] + -17.598;
   1:L PR[91] 10mm/sec CNT100;
   1:  PR[GP1:91,1] = PR[GP1:90,1] + -19.843;
   1:  PR[GP1:91,2] = PR[GP1:90,2] + -17.884;
   1:L PR[91] 10mm/sec CNT100;
   1:  PR[GP1:91,1] = PR[GP1:90,1] + -16.888;
   1:  PR[GP1:91,2] = PR[GP1:90,2] + -18.478;
   1:L PR[91] 10mm/sec CNT100;
   1:  PR[GP1:91,1] = PR[GP1:90,1] + -13.259;
   1:  PR[GP1:91,2] = PR[GP1:90,2] + -18.598;
   1:L PR[91] 10mm/sec CNT100;
   1:  PR[GP1:91,1] = PR[GP1:90,1] + -11.484;
   1:  PR[GP1:91,2] = PR[GP1:90,2] + -18.431;
   1:L PR[91] 10mm/sec CNT100;
   1:  PR[GP1:91,1] = PR[GP1:90,1] + -9.947;
   1:  PR[GP1:91,2] = PR[GP1:90,2] + -18.192;
   1:L PR[91] 10mm/sec CNT100;
   1:  PR[GP1:91,1] = PR[GP1:90,1] + -7.469;
   1:  PR[GP1:91,2] = PR[GP1:90,2] + -17.485;
   1:L PR[91] 10mm/sec CNT100;
   1:  PR[GP1:91,1] = PR[GP1:90,1] + -6.775;
   1:  PR[GP1:91,2] = PR[GP1:90,2] + -17.324;
   1:L PR[91] 10mm/sec CNT100;
   1:  PR[GP1:91,1] = PR[GP1:90,1] + -6.447;
   1:  PR[GP1:91,2] = PR[GP1:90,2] + -17.198;
   1:L PR[91] 10mm/sec CNT100;
   1:  PR[GP1:91,1] = PR[GP1:90,1] + -3.840;
   1:  PR[GP1:91,2] = PR[GP1:90,2] + -16.057;
   1:L PR[91] 10mm/sec CNT100;
   1:  PR[GP1:91,1] = PR[GP1:90,1] + -2.357;
   1:  PR[GP1:91,2] = PR[GP1:90,2] + -15.197;
   1:L PR[91] 10mm/sec CNT100;
   1:  PR[GP1:91,1] = PR[GP1:90,1] + -1.552;
   1:  PR[GP1:91,2] = PR[GP1:90,2] + -14.621;
   1:L PR[91] 10mm/sec CNT100;
   1:  PR[GP1:91,1] = PR[GP1:90,1] + -1.327;
   1:  PR[GP1:91,2] = PR[GP1:90,2] + -14.493;
   1:L PR[91] 10mm/sec CNT100;
   1:  PR[GP1:91,1] = PR[GP1:90,1] + -0.772;
   1:  PR[GP1:91,2] = PR[GP1:90,2] + -14.252;
   1:L PR[91] 10mm/sec CNT100;
   1:  PR[GP1:91,1] = PR[GP1:90,1] + -0.161;
   1:  PR[GP1:91,2] = PR[GP1:90,2] + -14.212;
   1:L PR[91] 10mm/sec CNT100;
   1:  PR[GP1:91,1] = PR[GP1:90,1] + 0.127;
   1:  PR[GP1:91,2] = PR[GP1:90,2] + -14.228;
   1:L PR[91] 10mm/sec CNT100;
   1:  PR[GP1:91,1] = PR[GP1:90,1] + 0.757;
   1:  PR[GP1:91,2] = PR[GP1:90,2] + -14.402;
   1:L PR[91] 10mm/sec CNT100;
   1:  PR[GP1:91,1] = PR[GP1:90,1] + 1.346;
   1:  PR[GP1:91,2] = PR[GP1:90,2] + -14.778;
   1:L PR[91] 10mm/sec CNT100;
   1:  PR[GP1:91,1] = PR[GP1:90,1] + 1.957;
   1:  PR[GP1:91,2] = PR[GP1:90,2] + -15.266;
   1:L PR[91] 10mm/sec CNT100;
   1:  PR[GP1:91,1] = PR[GP1:90,1] + 2.749;
   1:  PR[GP1:91,2] = PR[GP1:90,2] + -15.853;
   1:L PR[91] 10mm/sec CNT100;
   1:  PR[GP1:91,1] = PR[GP1:90,1] + 2.921;
   1:  PR[GP1:91,2] = PR[GP1:90,2] + -15.964;
   1:L PR[91] 10mm/sec CNT100;
   1:  PR[GP1:91,1] = PR[GP1:90,1] + 5.188;
   1:  PR[GP1:91,2] = PR[GP1:90,2] + -17.243;
   1:L PR[91] 10mm/sec CNT100;
   1:  PR[GP1:91,1] = PR[GP1:90,1] + 7.579;
   1:  PR[GP1:91,2] = PR[GP1:90,2] + -18.152;
   1:L PR[91] 10mm/sec CNT100;
   1:  PR[GP1:91,1] = PR[GP1:90,1] + 10.148;
   1:  PR[GP1:91,2] = PR[GP1:90,2] + -18.726;
   1:L PR[91] 10mm/sec CNT100;
   1:  PR[GP1:91,1] = PR[GP1:90,1] + 10.917;
   1:  PR[GP1:91,2] = PR[GP1:90,2] + -18.801;
   1:L PR[91] 10mm/sec CNT100;
   1:  PR[GP1:91,1] = PR[GP1:90,1] + 12.791;
   1:  PR[GP1:91,2] = PR[GP1:90,2] + -18.938;
   1:L PR[91] 10mm/sec CNT100;
   1:  PR[GP1:91,1] = PR[GP1:90,1] + 14.440;
   1:  PR[GP1:91,2] = PR[GP1:90,2] + -18.858;
   1:L PR[91] 10mm/sec CNT100;
   1:  PR[GP1:91,1] = PR[GP1:90,1] + 15.467;
   1:  PR[GP1:91,2] = PR[GP1:90,2] + -18.787;
   1:L PR[91] 10mm/sec CNT100;
   1:  PR[GP1:91,1] = PR[GP1:90,1] + 18.137;
   1:  PR[GP1:91,2] = PR[GP1:90,2] + -18.266;
   1:L PR[91] 10mm/sec CNT100;
   1:  PR[GP1:91,1] = PR[GP1:90,1] + 20.768;
   1:  PR[GP1:91,2] = PR[GP1:90,2] + -17.420;
   1:L PR[91] 10mm/sec CNT100;
   1:  PR[GP1:91,1] = PR[GP1:90,1] + 21.848;
   1:  PR[GP1:91,2] = PR[GP1:90,2] + -16.920;
   1:L PR[91] 10mm/sec CNT100;
   1:  PR[GP1:91,1] = PR[GP1:90,1] + 23.271;
   1:  PR[GP1:91,2] = PR[GP1:90,2] + -16.233;
   1:L PR[91] 10mm/sec CNT100;
   1:  PR[GP1:91,1] = PR[GP1:90,1] + 25.327;
   1:  PR[GP1:91,2] = PR[GP1:90,2] + -14.896;
   1:L PR[91] 10mm/sec CNT100;
   1:  PR[GP1:91,1] = PR[GP1:90,1] + 25.603;
   1:  PR[GP1:91,2] = PR[GP1:90,2] + -14.710;
   1:L PR[91] 10mm/sec CNT100;
   1:  PR[GP1:91,1] = PR[GP1:90,1] + 27.721;
   1:  PR[GP1:91,2] = PR[GP1:90,2] + -12.885;
   1:L PR[91] 10mm/sec CNT100;
   1:  PR[GP1:91,1] = PR[GP1:90,1] + 29.543;
   1:  PR[GP1:91,2] = PR[GP1:90,2] + -10.793;
   1:L PR[91] 10mm/sec CNT100;
   1:  PR[GP1:91,1] = PR[GP1:90,1] + 31.019;
   1:  PR[GP1:91,2] = PR[GP1:90,2] + -8.471;
   1:L PR[91] 10mm/sec CNT100;
   1:  PR[GP1:91,1] = PR[GP1:90,1] + 31.863;
   1:  PR[GP1:91,2] = PR[GP1:90,2] + -6.542;
   1:L PR[91] 10mm/sec CNT100;
   1:  PR[GP1:91,1] = PR[GP1:90,1] + 32.105;
   1:  PR[GP1:91,2] = PR[GP1:90,2] + -5.976;
   1:L PR[91] 10mm/sec CNT100;
   1:  PR[GP1:91,1] = PR[GP1:90,1] + 32.771;
   1:  PR[GP1:91,2] = PR[GP1:90,2] + -3.361;
   1:L PR[91] 10mm/sec CNT100;
   1:  PR[GP1:91,1] = PR[GP1:90,1] + 32.984;
   1:  PR[GP1:91,2] = PR[GP1:90,2] + -0.703;
   1:L PR[91] 10mm/sec CNT100;
   1:  PR[GP1:91,1] = PR[GP1:90,1] + 32.593;
   1:  PR[GP1:91,2] = PR[GP1:90,2] + 2.631;
   1:L PR[91] 10mm/sec CNT100;
   1:  PR[GP1:91,1] = PR[GP1:90,1] + 31.524;
   1:  PR[GP1:91,2] = PR[GP1:90,2] + 5.817;
   1:L PR[91] 10mm/sec CNT100;
   1:  PR[GP1:91,1] = PR[GP1:90,1] + 29.787;
   1:  PR[GP1:91,2] = PR[GP1:90,2] + 8.731;
   1:L PR[91] 10mm/sec CNT100;
   1:  PR[GP1:91,1] = PR[GP1:90,1] + 27.448;
   1:  PR[GP1:91,2] = PR[GP1:90,2] + 11.263;
   1:L PR[91] 10mm/sec CNT100;
   1:  PR[GP1:91,1] = PR[GP1:90,1] + 24.601;
   1:  PR[GP1:91,2] = PR[GP1:90,2] + 13.314;
   1:L PR[91] 10mm/sec CNT100;
   1:  PR[GP1:91,1] = PR[GP1:90,1] + 21.352;
   1:  PR[GP1:91,2] = PR[GP1:90,2] + 14.774;
   1:L PR[91] 10mm/sec CNT100;
   1:  PR[GP1:91,1] = PR[GP1:90,1] + 17.815;
   1:  PR[GP1:91,2] = PR[GP1:90,2] + 15.620;
   1:L PR[91] 10mm/sec CNT100;
   1:  PR[GP1:91,1] = PR[GP1:90,1] + 17.278;
   1:  PR[GP1:91,2] = PR[GP1:90,2] + 15.650;
   1:L PR[91] 10mm/sec CNT100;
   1:  PR[GP1:91,1] = PR[GP1:90,1] + 14.163;
   1:  PR[GP1:91,2] = PR[GP1:90,2] + 15.803;
   1:L PR[91] 10mm/sec CNT100;
   1:  PR[GP1:91,1] = PR[GP1:90,1] + 10.550;
   1:  PR[GP1:91,2] = PR[GP1:90,2] + 15.309;
   1:L PR[91] 10mm/sec CNT100;
   1:  PR[GP1:91,1] = PR[GP1:90,1] + 7.064;
   1:  PR[GP1:91,2] = PR[GP1:90,2] + 14.186;
   1:L PR[91] 10mm/sec CNT100;
   1:  PR[GP1:91,1] = PR[GP1:90,1] + 6.302;
   1:  PR[GP1:91,2] = PR[GP1:90,2] + 13.784;
   1:L PR[91] 10mm/sec CNT100;
   1:  PR[GP1:91,1] = PR[GP1:90,1] + 3.900;
   1:  PR[GP1:91,2] = PR[GP1:90,2] + 12.459;
   1:L PR[91] 10mm/sec CNT100;
   1:  PR[GP1:91,1] = PR[GP1:90,1] + 0.997;
   1:  PR[GP1:91,2] = PR[GP1:90,2] + 10.138;
   1:L PR[91] 10mm/sec CNT100;
   1:  PR[GP1:91,1] = PR[GP1:90,1] + 0.016;
   1:  PR[GP1:91,2] = PR[GP1:90,2] + 9.467;
   1:L PR[91] 10mm/sec CNT100;
   1:  PR[GP1:91,1] = PR[GP1:90,1] + -0.638;
   1:  PR[GP1:91,2] = PR[GP1:90,2] + 9.412;
   1:L PR[91] 10mm/sec CNT100;
   1:  PR[GP1:91,1] = PR[GP1:90,1] + -1.352;
   1:  PR[GP1:91,2] = PR[GP1:90,2] + 9.419;
   1:L PR[91] 10mm/sec CNT100;
   1:  PR[GP1:91,1] = PR[GP1:90,1] + -1.956;
   1:  PR[GP1:91,2] = PR[GP1:90,2] + 9.737;
   1:L PR[91] 10mm/sec CNT100;
   1:  PR[GP1:91,1] = PR[GP1:90,1] + -2.435;
   1:  PR[GP1:91,2] = PR[GP1:90,2] + 10.022;
   1:L PR[91] 10mm/sec CNT100;
   1:  PR[GP1:91,1] = PR[GP1:90,1] + -3.487;
   1:  PR[GP1:91,2] = PR[GP1:90,2] + 10.920;
   1:L PR[91] 10mm/sec CNT100;
   1:  PR[GP1:91,1] = PR[GP1:90,1] + -4.748;
   1:  PR[GP1:91,2] = PR[GP1:90,2] + 11.789;
   1:L PR[91] 10mm/sec CNT100;
   1:  PR[GP1:91,1] = PR[GP1:90,1] + -7.430;
   1:  PR[GP1:91,2] = PR[GP1:90,2] + 13.371;
   1:L PR[91] 10mm/sec CNT100;
   1:  PR[GP1:91,1] = PR[GP1:90,1] + -10.257;
   1:  PR[GP1:91,2] = PR[GP1:90,2] + 14.486;
   1:L PR[91] 10mm/sec CNT100;
   1:  PR[GP1:91,1] = PR[GP1:90,1] + -11.264;
   1:  PR[GP1:91,2] = PR[GP1:90,2] + 14.840;
   1:L PR[91] 10mm/sec CNT100;
   1:  PR[GP1:91,1] = PR[GP1:90,1] + -13.148;
   1:  PR[GP1:91,2] = PR[GP1:90,2] + 15.194;
   1:L PR[91] 10mm/sec CNT100;
   1:  PR[GP1:91,1] = PR[GP1:90,1] + -15.192;
   1:  PR[GP1:91,2] = PR[GP1:90,2] + 15.510;
   1:L PR[91] 10mm/sec CNT100;
   1:  PR[GP1:91,1] = PR[GP1:90,1] + -16.176;
   1:  PR[GP1:91,2] = PR[GP1:90,2] + 15.505;
   1:L PR[91] 10mm/sec CNT100;
   1:  PR[GP1:91,1] = PR[GP1:90,1] + -19.054;
   1:  PR[GP1:91,2] = PR[GP1:90,2] + 15.411;
   1:L PR[91] 10mm/sec CNT100;
   1:  PR[GP1:91,1] = PR[GP1:90,1] + -20.652;
   1:  PR[GP1:91,2] = PR[GP1:90,2] + 15.055;
   1:L PR[91] 10mm/sec CNT100;
   1:  PR[GP1:91,1] = PR[GP1:90,1] + -22.601;
   1:  PR[GP1:91,2] = PR[GP1:90,2] + 14.578;
   1:L PR[91] 10mm/sec CNT100;
   1:  PR[GP1:91,1] = PR[GP1:90,1] + -25.788;
   1:  PR[GP1:91,2] = PR[GP1:90,2] + 13.079;
   1:L PR[91] 10mm/sec CNT100;
   1:  PR[GP1:91,1] = PR[GP1:90,1] + -28.567;
   1:  PR[GP1:91,2] = PR[GP1:90,2] + 10.995;
   1:L PR[91] 10mm/sec CNT100;
   1:  PR[GP1:91,1] = PR[GP1:90,1] + -30.826;
   1:  PR[GP1:91,2] = PR[GP1:90,2] + 8.412;
   1:L PR[91] 10mm/sec CNT100;
   1:  PR[GP1:91,1] = PR[GP1:90,1] + -32.494;
   1:  PR[GP1:91,2] = PR[GP1:90,2] + 5.435;
   1:L PR[91] 10mm/sec CNT100;
   1:  PR[GP1:91,1] = PR[GP1:90,1] + -33.521;
   1:  PR[GP1:91,2] = PR[GP1:90,2] + 2.197;
   1:L PR[91] 10mm/sec CNT100;
   1:  PR[GP1:91,1] = PR[GP1:90,1] + -33.819;
   1:  PR[GP1:91,2] = PR[GP1:90,2] + -1.203;
   1:L PR[91] 10mm/sec CNT100;
   1:  PR[GP1:91,1] = PR[GP1:90,1] + -33.681;
   1:  PR[GP1:91,2] = PR[GP1:90,2] + -2.339;
   1:L PR[91] 10mm/sec CNT100;
   1:  PR[GP1:91,1] = PR[GP1:90,1] + -33.652;
   1:  PR[GP1:91,2] = PR[GP1:90,2] + -2.463;
   1:L PR[91] 10mm/sec CNT100;
   1:  PR[GP1:91,1] = PR[GP1:90,1] + -33.366;
   1:  PR[GP1:91,2] = PR[GP1:90,2] + -4.647;
   1:L PR[91] 10mm/sec CNT100;
   1:  PR[GP1:91,1] = PR[GP1:90,1] + -32.254;
   1:  PR[GP1:91,2] = PR[GP1:90,2] + -7.954;
   1:L PR[91] 10mm/sec CNT100;
   1:  PR[GP1:91,1] = PR[GP1:90,1] + -31.883;
   1:  PR[GP1:91,2] = PR[GP1:90,2] + -8.592;
   1:L PR[91] 10mm/sec CNT100;
   1:  PR[GP1:91,1] = PR[GP1:90,1] + -30.436;
   1:  PR[GP1:91,2] = PR[GP1:90,2] + -11.010;
   1:L PR[91] 10mm/sec CNT100;
   1:  PR[GP1:91,1] = PR[GP1:90,1] + -28.913;
   1:  PR[GP1:91,2] = PR[GP1:90,2] + -12.680;
   1:L PR[91] 10mm/sec CNT100;
   1:  PR[GP1:91,1] = PR[GP1:90,1] + -27.925;
   1:  PR[GP1:91,2] = PR[GP1:90,2] + -13.713;
   1:L PR[91] 10mm/sec CNT100;
   1:  PR[GP1:91,1] = PR[GP1:90,1] + -25.505;
   1:  PR[GP1:91,2] = PR[GP1:90,2] + -15.440;
   1:L PR[91] 10mm/sec CNT100;
   1:  PR[GP1:91,1] = PR[GP1:90,1] + -24.125;
   1:  PR[GP1:91,2] = PR[GP1:90,2] + -16.180;
   1:  PR[GP1:91,3] = PR[GP1:90,3] + 24.200;
   1:L PR[91] 10mm/sec CNT100;
   1:  PR[GP1:91,1] = PR[GP1:90,1] + -22.791;
   1:  PR[GP1:91,2] = PR[GP1:90,2] + -16.794;
   1:L PR[91] 10mm/sec CNT100;
   1:  PR[GP1:91,1] = PR[GP1:90,1] + -20.349;
   1:  PR[GP1:91,2] = PR[GP1:90,2] + -17.803;
   1:L PR[91] 10mm/sec CNT100;
   1:  PR[GP1:91,1] = PR[GP1:90,1] + -19.950;
   1:  PR[GP1:91,2] = PR[GP1:90,2] + -17.902;
   1:L PR[91] 10mm/sec CNT100;
   1:  PR[GP1:91,1] = PR[GP1:90,1] + -18.739;
   1:  PR[GP1:91,2] = PR[GP1:90,2] + -18.146;
   1:L PR[91] 10mm/sec CNT100;
   1:  PR[GP1:91,1] = PR[GP1:90,1] + -16.523;
   1:  PR[GP1:91,2] = PR[GP1:90,2] + -18.631;
   1:L PR[91] 10mm/sec CNT100;
   1:  PR[GP1:91,1] = PR[GP1:90,1] + -15.400;
   1:  PR[GP1:91,2] = PR[GP1:90,2] + -18.724;
   1:L PR[91] 10mm/sec CNT100;
   1:  PR[GP1:91,1] = PR[GP1:90,1] + -13.007;
   1:  PR[GP1:91,2] = PR[GP1:90,2] + -18.805;
   1:L PR[91] 10mm/sec CNT100;
   1:  PR[GP1:91,1] = PR[GP1:90,1] + -9.949;
   1:  PR[GP1:91,2] = PR[GP1:90,2] + -18.517;
   1:L PR[91] 10mm/sec CNT100;
   1:  PR[GP1:91,1] = PR[GP1:90,1] + -9.755;
   1:  PR[GP1:91,2] = PR[GP1:90,2] + -18.487;
   1:L PR[91] 10mm/sec CNT100;
   1:  PR[GP1:91,1] = PR[GP1:90,1] + -9.381;
   1:  PR[GP1:91,2] = PR[GP1:90,2] + -18.380;
   1:L PR[91] 10mm/sec CNT100;
   1:  PR[GP1:91,1] = PR[GP1:90,1] + -6.215;
   1:  PR[GP1:91,2] = PR[GP1:90,2] + -17.645;
   1:L PR[91] 10mm/sec CNT100;
   1:  PR[GP1:91,1] = PR[GP1:90,1] + -4.567;
   1:  PR[GP1:91,2] = PR[GP1:90,2] + -17.013;
   1:L PR[91] 10mm/sec CNT100;
   1:  PR[GP1:91,1] = PR[GP1:90,1] + -3.453;
   1:  PR[GP1:91,2] = PR[GP1:90,2] + -16.526;
   1:L PR[91] 10mm/sec CNT100;
   1:  PR[GP1:91,1] = PR[GP1:90,1] + -1.823;
   1:  PR[GP1:91,2] = PR[GP1:90,2] + -15.580;
   1:L PR[91] 10mm/sec CNT100;
   1:  PR[GP1:91,1] = PR[GP1:90,1] + -1.154;
   1:  PR[GP1:91,2] = PR[GP1:90,2] + -15.234;
   1:L PR[91] 10mm/sec CNT100;
   1:  PR[GP1:91,1] = PR[GP1:90,1] + -0.980;
   1:  PR[GP1:91,2] = PR[GP1:90,2] + -15.192;
   1:L PR[91] 10mm/sec CNT100;
   1:  PR[GP1:91,1] = PR[GP1:90,1] + -0.507;
   1:  PR[GP1:91,2] = PR[GP1:90,2] + -14.986;
   1:L PR[91] 10mm/sec CNT100;
   1:  PR[GP1:91,1] = PR[GP1:90,1] + 0.222;
   1:  PR[GP1:91,2] = PR[GP1:90,2] + -14.932;
   1:L PR[91] 10mm/sec CNT100;
   1:  PR[GP1:91,1] = PR[GP1:90,1] + 0.599;
   1:  PR[GP1:91,2] = PR[GP1:90,2] + -15.071;
   1:L PR[91] 10mm/sec CNT100;
   1:  PR[GP1:91,1] = PR[GP1:90,1] + 1.122;
   1:  PR[GP1:91,2] = PR[GP1:90,2] + -15.214;
   1:L PR[91] 10mm/sec CNT100;
   1:  PR[GP1:91,1] = PR[GP1:90,1] + 1.587;
   1:  PR[GP1:91,2] = PR[GP1:90,2] + -15.490;
   1:L PR[91] 10mm/sec CNT100;
   1:  PR[GP1:91,1] = PR[GP1:90,1] + 2.273;
   1:  PR[GP1:91,2] = PR[GP1:90,2] + -15.999;
   1:L PR[91] 10mm/sec CNT100;
   1:  PR[GP1:91,1] = PR[GP1:90,1] + 2.674;
   1:  PR[GP1:91,2] = PR[GP1:90,2] + -16.259;
   1:L PR[91] 10mm/sec CNT100;
   1:  PR[GP1:91,1] = PR[GP1:90,1] + 4.101;
   1:  PR[GP1:91,2] = PR[GP1:90,2] + -17.071;
   1:L PR[91] 10mm/sec CNT100;
   1:  PR[GP1:91,1] = PR[GP1:90,1] + 4.986;
   1:  PR[GP1:91,2] = PR[GP1:90,2] + -17.538;
   1:L PR[91] 10mm/sec CNT100;
   1:  PR[GP1:91,1] = PR[GP1:90,1] + 6.831;
   1:  PR[GP1:91,2] = PR[GP1:90,2] + -18.237;
   1:L PR[91] 10mm/sec CNT100;
   1:  PR[GP1:91,1] = PR[GP1:90,1] + 7.404;
   1:  PR[GP1:91,2] = PR[GP1:90,2] + -18.429;
   1:L PR[91] 10mm/sec CNT100;
   1:  PR[GP1:91,1] = PR[GP1:90,1] + 9.899;
   1:  PR[GP1:91,2] = PR[GP1:90,2] + -18.954;
   1:L PR[91] 10mm/sec CNT100;
   1:  PR[GP1:91,1] = PR[GP1:90,1] + 12.517;
   1:  PR[GP1:91,2] = PR[GP1:90,2] + -19.139;
   1:L PR[91] 10mm/sec CNT100;
   1:  PR[GP1:91,1] = PR[GP1:90,1] + 15.195;
   1:  PR[GP1:91,2] = PR[GP1:90,2] + -18.966;
   1:L PR[91] 10mm/sec CNT100;
   1:  PR[GP1:91,1] = PR[GP1:90,1] + 16.746;
   1:  PR[GP1:91,2] = PR[GP1:90,2] + -18.665;
   1:L PR[91] 10mm/sec CNT100;
   1:  PR[GP1:91,1] = PR[GP1:90,1] + 17.842;
   1:  PR[GP1:91,2] = PR[GP1:90,2] + -18.431;
   1:L PR[91] 10mm/sec CNT100;
   1:  PR[GP1:91,1] = PR[GP1:90,1] + 20.429;
   1:  PR[GP1:91,2] = PR[GP1:90,2] + -17.533;
   1:L PR[91] 10mm/sec CNT100;
   1:  PR[GP1:91,1] = PR[GP1:90,1] + 22.924;
   1:  PR[GP1:91,2] = PR[GP1:90,2] + -16.326;
   1:L PR[91] 10mm/sec CNT100;
   1:  PR[GP1:91,1] = PR[GP1:90,1] + 23.920;
   1:  PR[GP1:91,2] = PR[GP1:90,2] + -15.679;
   1:L PR[91] 10mm/sec CNT100;
   1:  PR[GP1:91,1] = PR[GP1:90,1] + 25.234;
   1:  PR[GP1:91,2] = PR[GP1:90,2] + -14.797;
   1:L PR[91] 10mm/sec CNT100;
   1:  PR[GP1:91,1] = PR[GP1:90,1] + 27.011;
   1:  PR[GP1:91,2] = PR[GP1:90,2] + -13.235;
   1:L PR[91] 10mm/sec CNT100;
   1:  PR[GP1:91,1] = PR[GP1:90,1] + 27.314;
   1:  PR[GP1:91,2] = PR[GP1:90,2] + -12.961;
   1:L PR[91] 10mm/sec CNT100;
   1:  PR[GP1:91,1] = PR[GP1:90,1] + 29.118;
   1:  PR[GP1:91,2] = PR[GP1:90,2] + -10.856;
   1:L PR[91] 10mm/sec CNT100;
   1:  PR[GP1:91,1] = PR[GP1:90,1] + 30.581;
   1:  PR[GP1:91,2] = PR[GP1:90,2] + -8.534;
   1:L PR[91] 10mm/sec CNT100;
   1:  PR[GP1:91,1] = PR[GP1:90,1] + 31.030;
   1:  PR[GP1:91,2] = PR[GP1:90,2] + -7.506;
   1:L PR[91] 10mm/sec CNT100;
   1:  PR[GP1:91,1] = PR[GP1:90,1] + 31.656;
   1:  PR[GP1:91,2] = PR[GP1:90,2] + -6.043;
   1:L PR[91] 10mm/sec CNT100;
   1:  PR[GP1:91,1] = PR[GP1:90,1] + 32.314;
   1:  PR[GP1:91,2] = PR[GP1:90,2] + -3.435;
   1:L PR[91] 10mm/sec CNT100;
   1:  PR[GP1:91,1] = PR[GP1:90,1] + 32.524;
   1:  PR[GP1:91,2] = PR[GP1:90,2] + -0.777;
   1:L PR[91] 10mm/sec CNT100;
   1:  PR[GP1:91,1] = PR[GP1:90,1] + 32.134;
   1:  PR[GP1:91,2] = PR[GP1:90,2] + 2.567;
   1:L PR[91] 10mm/sec CNT100;
   1:  PR[GP1:91,1] = PR[GP1:90,1] + 31.059;
   1:  PR[GP1:91,2] = PR[GP1:90,2] + 5.755;
   1:L PR[91] 10mm/sec CNT100;
   1:  PR[GP1:91,1] = PR[GP1:90,1] + 29.316;
   1:  PR[GP1:91,2] = PR[GP1:90,2] + 8.670;
   1:L PR[91] 10mm/sec CNT100;
   1:  PR[GP1:91,1] = PR[GP1:90,1] + 26.972;
   1:  PR[GP1:91,2] = PR[GP1:90,2] + 11.201;
   1:L PR[91] 10mm/sec CNT100;
   1:  PR[GP1:91,1] = PR[GP1:90,1] + 24.120;
   1:  PR[GP1:91,2] = PR[GP1:90,2] + 13.224;
   1:L PR[91] 10mm/sec CNT100;
   1:  PR[GP1:91,1] = PR[GP1:90,1] + 20.864;
   1:  PR[GP1:91,2] = PR[GP1:90,2] + 14.683;
   1:L PR[91] 10mm/sec CNT100;
   1:  PR[GP1:91,1] = PR[GP1:90,1] + 17.339;
   1:  PR[GP1:91,2] = PR[GP1:90,2] + 15.522;
   1:L PR[91] 10mm/sec CNT100;
   1:  PR[GP1:91,1] = PR[GP1:90,1] + 13.709;
   1:  PR[GP1:91,2] = PR[GP1:90,2] + 15.689;
   1:L PR[91] 10mm/sec CNT100;
   1:  PR[GP1:91,1] = PR[GP1:90,1] + 10.089;
   1:  PR[GP1:91,2] = PR[GP1:90,2] + 15.198;
   1:L PR[91] 10mm/sec CNT100;
   1:  PR[GP1:91,1] = PR[GP1:90,1] + 7.730;
   1:  PR[GP1:91,2] = PR[GP1:90,2] + 14.439;
   1:L PR[91] 10mm/sec CNT100;
   1:  PR[GP1:91,1] = PR[GP1:90,1] + 6.635;
   1:  PR[GP1:91,2] = PR[GP1:90,2] + 14.071;
   1:L PR[91] 10mm/sec CNT100;
   1:  PR[GP1:91,1] = PR[GP1:90,1] + 3.470;
   1:  PR[GP1:91,2] = PR[GP1:90,2] + 12.336;
   1:L PR[91] 10mm/sec CNT100;
   1:  PR[GP1:91,1] = PR[GP1:90,1] + 1.024;
   1:  PR[GP1:91,2] = PR[GP1:90,2] + 10.401;
   1:L PR[91] 10mm/sec CNT100;
   1:  PR[GP1:91,1] = PR[GP1:90,1] + 0.509;
   1:  PR[GP1:91,2] = PR[GP1:90,2] + 10.144;
   1:L PR[91] 10mm/sec CNT100;
   1:  PR[GP1:91,1] = PR[GP1:90,1] + 0.042;
   1:  PR[GP1:91,2] = PR[GP1:90,2] + 9.823;
   1:L PR[91] 10mm/sec CNT100;
   1:  PR[GP1:91,1] = PR[GP1:90,1] + -0.358;
   1:  PR[GP1:91,2] = PR[GP1:90,2] + 9.790;
   1:L PR[91] 10mm/sec CNT100;
   1:  PR[GP1:91,1] = PR[GP1:90,1] + -1.329;
   1:  PR[GP1:91,2] = PR[GP1:90,2] + 9.799;
   1:L PR[91] 10mm/sec CNT100;
   1:  PR[GP1:91,1] = PR[GP1:90,1] + -2.282;
   1:  PR[GP1:91,2] = PR[GP1:90,2] + 10.309;
   1:L PR[91] 10mm/sec CNT100;
   1:  PR[GP1:91,1] = PR[GP1:90,1] + -2.517;
   1:  PR[GP1:91,2] = PR[GP1:90,2] + 10.510;
   1:L PR[91] 10mm/sec CNT100;
   1:  PR[GP1:91,1] = PR[GP1:90,1] + -4.639;
   1:  PR[GP1:91,2] = PR[GP1:90,2] + 11.972;
   1:L PR[91] 10mm/sec CNT100;
   1:  PR[GP1:91,1] = PR[GP1:90,1] + -6.433;
   1:  PR[GP1:91,2] = PR[GP1:90,2] + 13.031;
   1:L PR[91] 10mm/sec CNT100;
   1:  PR[GP1:91,1] = PR[GP1:90,1] + -7.318;
   1:  PR[GP1:91,2] = PR[GP1:90,2] + 13.434;
   1:L PR[91] 10mm/sec CNT100;
   1:  PR[GP1:91,1] = PR[GP1:90,1] + -9.506;
   1:  PR[GP1:91,2] = PR[GP1:90,2] + 14.239;
   1:L PR[91] 10mm/sec CNT100;
   1:  PR[GP1:91,1] = PR[GP1:90,1] + -10.650;
   1:  PR[GP1:91,2] = PR[GP1:90,2] + 14.676;
   1:L PR[91] 10mm/sec CNT100;
   1:  PR[GP1:91,1] = PR[GP1:90,1] + -13.259;
   1:  PR[GP1:91,2] = PR[GP1:90,2] + 15.167;
   1:L PR[91] 10mm/sec CNT100;
   1:  PR[GP1:91,1] = PR[GP1:90,1] + -14.598;
   1:  PR[GP1:91,2] = PR[GP1:90,2] + 15.374;
   1:L PR[91] 10mm/sec CNT100;
   1:  PR[GP1:91,1] = PR[GP1:90,1] + -16.274;
   1:  PR[GP1:91,2] = PR[GP1:90,2] + 15.366;
   1:L PR[91] 10mm/sec CNT100;
   1:  PR[GP1:91,1] = PR[GP1:90,1] + -18.495;
   1:  PR[GP1:91,2] = PR[GP1:90,2] + 15.293;
   1:L PR[91] 10mm/sec CNT100;
   1:  PR[GP1:91,1] = PR[GP1:90,1] + -19.341;
   1:  PR[GP1:91,2] = PR[GP1:90,2] + 15.122;
   1:L PR[91] 10mm/sec CNT100;
   1:  PR[GP1:91,1] = PR[GP1:90,1] + -22.176;
   1:  PR[GP1:91,2] = PR[GP1:90,2] + 14.479;
   1:L PR[91] 10mm/sec CNT100;
   1:  PR[GP1:91,1] = PR[GP1:90,1] + -23.966;
   1:  PR[GP1:91,2] = PR[GP1:90,2] + 13.688;
   1:L PR[91] 10mm/sec CNT100;
   1:  PR[GP1:91,1] = PR[GP1:90,1] + -25.443;
   1:  PR[GP1:91,2] = PR[GP1:90,2] + 12.995;
   1:L PR[91] 10mm/sec CNT100;
   1:  PR[GP1:91,1] = PR[GP1:90,1] + -28.230;
   1:  PR[GP1:91,2] = PR[GP1:90,2] + 10.909;
   1:L PR[91] 10mm/sec CNT100;
   1:  PR[GP1:91,1] = PR[GP1:90,1] + -30.495;
   1:  PR[GP1:91,2] = PR[GP1:90,2] + 8.322;
   1:L PR[91] 10mm/sec CNT100;
   1:  PR[GP1:91,1] = PR[GP1:90,1] + -32.167;
   1:  PR[GP1:91,2] = PR[GP1:90,2] + 5.340;
   1:L PR[91] 10mm/sec CNT100;
   1:  PR[GP1:91,1] = PR[GP1:90,1] + -33.198;
   1:  PR[GP1:91,2] = PR[GP1:90,2] + 2.096;
   1:L PR[91] 10mm/sec CNT100;
   1:  PR[GP1:91,1] = PR[GP1:90,1] + -33.497;
   1:  PR[GP1:91,2] = PR[GP1:90,2] + -1.306;
   1:L PR[91] 10mm/sec CNT100;
   1:  PR[GP1:91,1] = PR[GP1:90,1] + -33.035;
   1:  PR[GP1:91,2] = PR[GP1:90,2] + -4.766;
   1:L PR[91] 10mm/sec CNT100;
   1:  PR[GP1:91,1] = PR[GP1:90,1] + -31.917;
   1:  PR[GP1:91,2] = PR[GP1:90,2] + -8.082;
   1:L PR[91] 10mm/sec CNT100;
   1:  PR[GP1:91,1] = PR[GP1:90,1] + -31.826;
   1:  PR[GP1:91,2] = PR[GP1:90,2] + -8.238;
   1:L PR[91] 10mm/sec CNT100;
   1:  PR[GP1:91,1] = PR[GP1:90,1] + -30.937;
   1:  PR[GP1:91,2] = PR[GP1:90,2] + -9.724;
   1:L PR[91] 10mm/sec CNT100;
   1:  PR[GP1:91,1] = PR[GP1:90,1] + -30.031;
   1:  PR[GP1:91,2] = PR[GP1:90,2] + -11.162;
   1:L PR[91] 10mm/sec CNT100;
   1:  PR[GP1:91,1] = PR[GP1:90,1] + -27.968;
   1:  PR[GP1:91,2] = PR[GP1:90,2] + -13.338;
   1:L PR[91] 10mm/sec CNT100;
   1:  PR[GP1:91,1] = PR[GP1:90,1] + -27.383;
   1:  PR[GP1:91,2] = PR[GP1:90,2] + -13.921;
   1:L PR[91] 10mm/sec CNT100;
   1:  PR[GP1:91,1] = PR[GP1:90,1] + -25.491;
   1:  PR[GP1:91,2] = PR[GP1:90,2] + -15.272;
   1:L PR[91] 10mm/sec CNT100;
   1:  PR[GP1:91,1] = PR[GP1:90,1] + -23.536;
   1:  PR[GP1:91,2] = PR[GP1:90,2] + -16.395;
   1:  PR[GP1:91,3] = PR[GP1:90,3] + 25.300;
   1:L PR[91] 10mm/sec CNT100;
   1:  PR[GP1:91,1] = PR[GP1:90,1] + -22.844;
   1:  PR[GP1:91,2] = PR[GP1:90,2] + -16.713;
   1:L PR[91] 10mm/sec CNT100;
   1:  PR[GP1:91,1] = PR[GP1:90,1] + -19.801;
   1:  PR[GP1:91,2] = PR[GP1:90,2] + -17.973;
   1:L PR[91] 10mm/sec CNT100;
   1:  PR[GP1:91,1] = PR[GP1:90,1] + -19.408;
   1:  PR[GP1:91,2] = PR[GP1:90,2] + -18.076;
   1:L PR[91] 10mm/sec CNT100;
   1:  PR[GP1:91,1] = PR[GP1:90,1] + -16.203;
   1:  PR[GP1:91,2] = PR[GP1:90,2] + -18.778;
   1:L PR[91] 10mm/sec CNT100;
   1:  PR[GP1:91,1] = PR[GP1:90,1] + -13.820;
   1:  PR[GP1:91,2] = PR[GP1:90,2] + -18.976;
   1:L PR[91] 10mm/sec CNT100;
   1:  PR[GP1:91,1] = PR[GP1:90,1] + -12.755;
   1:  PR[GP1:91,2] = PR[GP1:90,2] + -19.012;
   1:L PR[91] 10mm/sec CNT100;
   1:  PR[GP1:91,1] = PR[GP1:90,1] + -11.071;
   1:  PR[GP1:91,2] = PR[GP1:90,2] + -18.854;
   1:L PR[91] 10mm/sec CNT100;
   1:  PR[GP1:91,1] = PR[GP1:90,1] + -9.033;
   1:  PR[GP1:91,2] = PR[GP1:90,2] + -18.730;
   1:L PR[91] 10mm/sec CNT100;
   1:  PR[GP1:91,1] = PR[GP1:90,1] + -7.667;
   1:  PR[GP1:91,2] = PR[GP1:90,2] + -18.433;
   1:L PR[91] 10mm/sec CNT100;
   1:  PR[GP1:91,1] = PR[GP1:90,1] + -5.654;
   1:  PR[GP1:91,2] = PR[GP1:90,2] + -17.966;
   1:L PR[91] 10mm/sec CNT100;
   1:  PR[GP1:91,1] = PR[GP1:90,1] + -3.430;
   1:  PR[GP1:91,2] = PR[GP1:90,2] + -17.113;
   1:L PR[91] 10mm/sec CNT100;
   1:  PR[GP1:91,1] = PR[GP1:90,1] + -2.970;
   1:  PR[GP1:91,2] = PR[GP1:90,2] + -16.960;
   1:L PR[91] 10mm/sec CNT100;
   1:  PR[GP1:91,1] = PR[GP1:90,1] + -0.847;
   1:  PR[GP1:91,2] = PR[GP1:90,2] + -15.880;
   1:L PR[91] 10mm/sec CNT100;
